LIN {X 0.019,Y -212.975,Z 813.838,A 0.000,B 0.000,C 90.000,E1 330.845} C_DIS
LIN {X 0.093,Y -220.835,Z 813.816,A 0.000,B 0.000,C 90.000,E1 326.914} C_DIS
LIN {X -0.032,Y -227.717,Z 813.799,A 0.000,B 0.000,C 90.000,E1 323.863} C_DIS
LIN {X 0.055,Y -235.033,Z 813.782,A 0.000,B 0.000,C 90.000,E1 320.803} C_DIS
LIN {X -0.068,Y -244.076,Z 813.764,A 0.000,B 0.000,C 90.000,E1 317.472} C_DIS
LIN {X -0.126,Y -253.936,Z 813.745,A 0.000,B 0.000,C 90.000,E1 314.190} C_DIS
LIN {X -0.103,Y -263.291,Z 813.729,A 0.000,B 0.000,C 90.000,E1 311.310} C_DIS
LIN {X 0.023,Y -275.912,Z 813.710,A 0.000,B 0.000,C 90.000,E1 307.764} C_DIS
LIN {X -0.077,Y -288.380,Z 813.693,A 0.000,B 0.000,C 90.000,E1 304.692} C_DIS
LIN {X -0.096,Y -300.556,Z 813.678,A 0.000,B 0.000,C 90.000,E1 302.005} C_DIS
LIN {X 0.089,Y -312.158,Z 813.665,A 0.000,B 0.000,C 90.000,E1 299.667} C_DIS
LIN {X -0.018,Y -328.621,Z 813.649,A 0.000,B 0.000,C 90.000,E1 296.796} C_DIS
LIN {X 0.198,Y -346.426,Z 813.633,A 0.000,B 0.000,C 90.000,E1 293.951} C_DIS
LIN {X 0.036,Y -359.385,Z 813.623,A 0.000,B 0.000,C 90.000,E1 292.153} C_DIS
LIN {X 0.081,Y -375.773,Z 813.612,A 0.000,B 0.000,C 90.000,E1 290.066} C_DIS
LIN {X -0.012,Y -393.420,Z 813.600,A 0.000,B 0.000,C 90.000,E1 288.055} C_DIS
LIN {X -0.013,Y -411.061,Z 813.590,A 0.000,B 0.000,C 90.000,E1 286.134} C_DIS
LIN {X 0.036,Y -423.562,Z 813.582,A 0.000,B 0.000,C 90.000,E1 284.773} C_DIS
LIN {X 0.129,Y -435.900,Z 813.575,A 0.000,B 0.000,C 90.000,E1 283.411} C_DIS
LIN {X 0.080,Y -445.463,Z 813.569,A 0.000,B 0.000,C 90.000,E1 282.355} C_DIS
LIN {X -0.139,Y -456.594,Z 813.561,A 0.000,B 0.000,C 90.000,E1 281.074} C_DIS
LIN {X 0.054,Y -464.756,Z 813.556,A 0.000,B 0.000,C 90.000,E1 280.018} C_DIS
LIN {X -0.204,Y -472.214,Z 813.550,A 0.000,B 0.000,C 90.000,E1 279.029} C_DIS
LIN {X 0.228,Y -477.257,Z 813.546,A 0.000,B 0.000,C 90.000,E1 278.219} C_DIS
LIN {X 0.169,Y -481.626,Z 813.542,A 0.000,B 0.000,C 90.000,E1 277.473} C_DIS
LIN {X 0.218,Y -485.397,Z 813.537,A 0.000,B 0.000,C 90.000,E1 276.720} C_DIS
LIN {X -0.195,Y -488.429,Z 813.533,A 0.000,B 0.000,C 90.000,E1 276.024} C_DIS
LIN {X -0.042,Y -490.064,Z 813.531,A 0.000,B 0.000,C 90.000,E1 275.511} C_DIS
LIN {X 0.172,Y -491.281,Z 813.528,A 0.000,B 0.000,C 90.000,E1 274.992} C_DIS
LIN {X -0.095,Y -492.106,Z 813.525,A 0.000,B 0.000,C 90.000,E1 274.531} C_DIS
LIN {X 0.133,Y -492.547,Z 813.522,A 0.000,B 0.000,C 90.000,E1 274.012} C_DIS
LIN {X -0.160,Y -492.648,Z 813.520,A 0.000,B 0.000,C 90.000,E1 273.555} C_DIS
LIN {X 0.072,Y -492.322,Z 813.517,A 0.000,B 0.000,C 90.000,E1 273.037} C_DIS
LIN {X -0.213,Y -491.589,Z 813.514,A 0.000,B 0.000,C 90.000,E1 272.579} C_DIS
LIN {X -0.007,Y -490.500,Z 813.511,A 0.000,B 0.000,C 90.000,E1 272.064} C_DIS
LIN {X 0.211,Y -488.923,Z 813.509,A 0.000,B 0.000,C 90.000,E1 271.547} C_DIS
LIN {X -0.082,Y -486.963,Z 813.506,A 0.000,B 0.000,C 90.000,E1 271.088} C_DIS
LIN {X 0.106,Y -484.457,Z 813.503,A 0.000,B 0.000,C 90.000,E1 270.573} C_DIS
LIN {X -0.207,Y -481.352,Z 813.500,A 0.000,B 0.000,C 90.000,E1 270.115} C_DIS
LIN {X -0.053,Y -477.541,Z 813.498,A 0.000,B 0.000,C 90.000,E1 269.599} C_DIS
LIN {X 0.077,Y -472.892,Z 813.495,A 0.000,B 0.000,C 90.000,E1 269.083} C_DIS
LIN {X 0.214,Y -467.213,Z 813.492,A 0.000,B 0.000,C 90.000,E1 268.568} C_DIS
LIN {X -0.189,Y -464.243,Z 813.491,A 0.000,B 0.000,C 90.000,E1 268.396} C_DIS
LIN {X -0.213,Y -457.716,Z 813.489,A 0.000,B 0.000,C 90.000,E1 267.993} C_DIS
LIN {X -0.131,Y -450.659,Z 813.487,A 0.000,B 0.000,C 90.000,E1 267.650} C_DIS
LIN {X 0.053,Y -442.949,Z 813.485,A 0.000,B 0.000,C 90.000,E1 267.364} C_DIS
LIN {X -0.148,Y -434.987,Z 813.484,A 0.000,B 0.000,C 90.000,E1 267.192} C_DIS
LIN {X 0.170,Y -427.099,Z 813.484,A 0.000,B 0.000,C 90.000,E1 267.020} C_DIS
LIN {X 0.184,Y -419.177,Z 813.483,A 0.000,B 0.000,C 90.000,E1 266.963} C_DIS
LIN {X 0.051,Y -180.989,Z 813.483,A 0.000,B 0.000,C 90.000,E1 266.963} C_DIS
LIN {X -0.017,Y -180.848,Z 813.472,A 0.000,B 0.000,C 90.000,E1 264.951} C_DIS
LIN {X 0.066,Y -178.958,Z 813.444,A 0.000,B 0.000,C 90.000,E1 259.859} C_DIS
LIN {X -0.043,Y -177.363,Z 813.430,A 0.000,B 0.000,C 90.000,E1 257.353} C_DIS
LIN {X 0.053,Y -175.535,Z 813.411,A 0.000,B 0.000,C 90.000,E1 253.921} C_DIS
LIN {X 0.054,Y -172.270,Z 813.387,A 0.000,B 0.000,C 90.000,E1 249.645} C_DIS
LIN {X 0.093,Y -171.749,Z 813.382,A 0.000,B 0.000,C 90.000,E1 248.773} C_DIS
LIN {X -0.050,Y -167.346,Z 813.353,A 0.000,B 0.000,C 90.000,E1 243.640} C_DIS
LIN {X 0.032,Y -166.734,Z 813.349,A 0.000,B 0.000,C 90.000,E1 242.743} C_DIS
LIN {X -0.055,Y -162.714,Z 813.324,A 0.000,B 0.000,C 90.000,E1 238.408} C_DIS
LIN {X 0.006,Y -161.404,Z 813.315,A 0.000,B 0.000,C 90.000,E1 236.628} C_DIS
LIN {X 0.048,Y -157.396,Z 813.290,A 0.000,B 0.000,C 90.000,E1 232.190} C_DIS
LIN {X -0.019,Y -155.394,Z 813.275,A 0.000,B 0.000,C 90.000,E1 229.542} C_DIS
LIN {X 0.021,Y -151.727,Z 813.250,A 0.000,B 0.000,C 90.000,E1 225.040} C_DIS
LIN {X 0.037,Y -149.923,Z 813.235,A 0.000,B 0.000,C 90.000,E1 222.324} C_DIS
LIN {X -0.046,Y -146.775,Z 813.210,A 0.000,B 0.000,C 90.000,E1 217.810} C_DIS
LIN {X 0.058,Y -145.346,Z 813.195,A 0.000,B 0.000,C 90.000,E1 215.025} C_DIS
LIN {X -0.027,Y -142.420,Z 813.164,A 0.000,B 0.000,C 90.000,E1 209.539} C_DIS
LIN {X 0.022,Y -141.407,Z 813.149,A 0.000,B 0.000,C 90.000,E1 206.744} C_DIS
LIN {X 0.009,Y -139.358,Z 813.112,A 0.000,B 0.000,C 90.000,E1 200.248} C_DIS
LIN {X -0.002,Y -138.799,Z 813.097,A 0.000,B 0.000,C 90.000,E1 197.457} C_DIS
LIN {X 0.052,Y -138.348,Z 813.055,A 0.000,B 0.000,C 90.000,E1 189.962} C_DIS
LIN {X 0.070,Y -139.370,Z 813.009,A 0.000,B 0.000,C 90.000,E1 181.547} C_DIS
LIN {X -0.016,Y -141.258,Z 812.973,A 0.000,B 0.000,C 90.000,E1 175.065} C_DIS
LIN {X -0.058,Y -142.626,Z 812.957,A 0.000,B 0.000,C 90.000,E1 172.299} C_DIS
LIN {X 0.035,Y -144.948,Z 812.931,A 0.000,B 0.000,C 90.000,E1 167.645} C_DIS
LIN {X 0.026,Y -147.577,Z 812.911,A 0.000,B 0.000,C 90.000,E1 163.976} C_DIS
LIN {X -0.085,Y -150.189,Z 812.891,A 0.000,B 0.000,C 90.000,E1 160.369} C_DIS
LIN {X -0.077,Y -153.568,Z 812.871,A 0.000,B 0.000,C 90.000,E1 156.741} C_DIS
LIN {X -0.026,Y -156.985,Z 812.851,A 0.000,B 0.000,C 90.000,E1 153.127} C_DIS
LIN {X 0.047,Y -161.098,Z 812.831,A 0.000,B 0.000,C 90.000,E1 149.537} C_DIS
LIN {X -0.007,Y -163.201,Z 812.821,A 0.000,B 0.000,C 90.000,E1 147.788} C_DIS
LIN {X -0.002,Y -167.628,Z 812.802,A 0.000,B 0.000,C 90.000,E1 144.276} C_DIS
LIN {X 0.013,Y -171.455,Z 812.787,A 0.000,B 0.000,C 90.000,E1 141.662} C_DIS
LIN {X -0.056,Y -176.379,Z 812.768,A 0.000,B 0.000,C 90.000,E1 138.243} C_DIS
LIN {X 0.066,Y -180.671,Z 812.754,A 0.000,B 0.000,C 90.000,E1 135.648} C_DIS
LIN {X 0.048,Y -186.074,Z 812.735,A 0.000,B 0.000,C 90.000,E1 132.285} C_DIS
LIN {X -0.015,Y -190.711,Z 812.721,A 0.000,B 0.000,C 90.000,E1 129.806} C_DIS
LIN {X 0.035,Y -192.711,Z 812.714,A 0.000,B 0.000,C 90.000,E1 128.588} C_DIS
LIN {X 0.010,Y -293.159,Z 812.714,A 0.000,B 0.000,C 90.000,E1 128.588} C_DIS
LIN {X -0.075,Y -294.254,Z 812.714,A 0.000,B 0.000,C 90.000,E1 128.588} C_DIS
LIN {X -0.110,Y -299.039,Z 812.713,A 0.000,B 0.000,C 90.000,E1 128.382} C_DIS
LIN {X -0.143,Y -301.560,Z 812.712,A 0.000,B 0.000,C 90.000,E1 128.177} C_DIS
LIN {X 0.042,Y -305.369,Z 812.709,A 0.000,B 0.000,C 90.000,E1 127.649} C_DIS
LIN {X 0.053,Y -307.140,Z 812.707,A 0.000,B 0.000,C 90.000,E1 127.317} C_DIS
LIN {X 0.006,Y -308.524,Z 812.706,A 0.000,B 0.000,C 90.000,E1 126.996} C_DIS
LIN {X -0.054,Y -316.443,Z 812.691,A 0.000,B 0.000,C 90.000,E1 124.405} C_DIS
LIN {X -0.054,Y -327.496,Z 812.673,A 0.000,B 0.000,C 90.000,E1 121.209} C_DIS
LIN {X 0.114,Y -338.834,Z 812.658,A 0.000,B 0.000,C 90.000,E1 118.359} C_DIS
LIN {X 0.122,Y -351.598,Z 812.642,A 0.000,B 0.000,C 90.000,E1 115.591} C_DIS
LIN {X -0.026,Y -364.229,Z 812.629,A 0.000,B 0.000,C 90.000,E1 113.206} C_DIS
LIN {X -0.008,Y -378.165,Z 812.616,A 0.000,B 0.000,C 90.000,E1 110.844} C_DIS
LIN {X -0.045,Y -393.504,Z 812.603,A 0.000,B 0.000,C 90.000,E1 108.544} C_DIS
LIN {X 0.190,Y -410.357,Z 812.590,A 0.000,B 0.000,C 90.000,E1 106.260} C_DIS
LIN {X -0.190,Y -428.847,Z 812.578,A 0.000,B 0.000,C 90.000,E1 104.120} C_DIS
LIN {X -0.052,Y -448.726,Z 812.567,A 0.000,B 0.000,C 90.000,E1 102.007} C_DIS
LIN {X -0.001,Y -466.598,Z 812.557,A 0.000,B 0.000,C 90.000,E1 100.310} C_DIS
LIN {X 0.023,Y -468.920,Z 812.556,A 0.000,B 0.000,C 90.000,E1 100.074} C_DIS
LIN {X -0.160,Y -470.769,Z 812.555,A 0.000,B 0.000,C 90.000,E1 99.849} C_DIS
LIN {X 0.202,Y -472.166,Z 812.553,A 0.000,B 0.000,C 90.000,E1 99.557} C_DIS
LIN {X -0.163,Y -473.990,Z 812.550,A 0.000,B 0.000,C 90.000,E1 99.095} C_DIS
LIN {X 0.022,Y -474.720,Z 812.548,A 0.000,B 0.000,C 90.000,E1 98.568} C_DIS
LIN {X 0.146,Y -474.481,Z 812.545,A 0.000,B 0.000,C 90.000,E1 98.049} C_DIS
LIN {X -0.193,Y -473.242,Z 812.542,A 0.000,B 0.000,C 90.000,E1 97.587} C_DIS
LIN {X 0.136,Y -472.188,Z 812.541,A 0.000,B 0.000,C 90.000,E1 97.296} C_DIS
LIN {X -0.063,Y -470.775,Z 812.539,A 0.000,B 0.000,C 90.000,E1 97.068} C_DIS
LIN {X 0.086,Y -453.158,Z 812.524,A 0.000,B 0.000,C 90.000,E1 94.245} C_DIS
LIN {X 0.028,Y -444.098,Z 812.515,A 0.000,B 0.000,C 90.000,E1 92.694} C_DIS
LIN {X -0.045,Y -433.373,Z 812.505,A 0.000,B 0.000,C 90.000,E1 90.859} C_DIS
LIN {X -0.041,Y -423.794,Z 812.496,A 0.000,B 0.000,C 90.000,E1 89.255} C_DIS
LIN {X -0.192,Y -414.104,Z 812.487,A 0.000,B 0.000,C 90.000,E1 87.650} C_DIS
LIN {X -0.104,Y -404.224,Z 812.478,A 0.000,B 0.000,C 90.000,E1 85.988} C_DIS
LIN {X -0.056,Y -391.053,Z 812.465,A 0.000,B 0.000,C 90.000,E1 83.742} C_DIS
LIN {X 0.110,Y -378.181,Z 812.453,A 0.000,B 0.000,C 90.000,E1 81.432} C_DIS
LIN {X 0.059,Y -364.163,Z 812.438,A 0.000,B 0.000,C 90.000,E1 78.814} C_DIS
LIN {X 0.132,Y -350.810,Z 812.423,A 0.000,B 0.000,C 90.000,E1 76.117} C_DIS
LIN {X -0.134,Y -340.550,Z 812.411,A 0.000,B 0.000,C 90.000,E1 74.031} C_DIS
LIN {X 0.111,Y -328.959,Z 812.397,A 0.000,B 0.000,C 90.000,E1 71.511} C_DIS
LIN {X 0.091,Y -316.298,Z 812.382,A 0.000,B 0.000,C 90.000,E1 68.666} C_DIS
LIN {X 0.067,Y -302.768,Z 812.364,A 0.000,B 0.000,C 90.000,E1 65.433} C_DIS
LIN {X -0.116,Y -290.215,Z 812.345,A 0.000,B 0.000,C 90.000,E1 62.153} C_DIS
LIN {X 0.070,Y -280.606,Z 812.330,A 0.000,B 0.000,C 90.000,E1 59.410} C_DIS
LIN {X 0.127,Y -270.334,Z 812.313,A 0.000,B 0.000,C 90.000,E1 56.294} C_DIS
LIN {X 0.016,Y -262.692,Z 812.299,A 0.000,B 0.000,C 90.000,E1 53.863} C_DIS
LIN {X -0.023,Y -256.222,Z 812.287,A 0.000,B 0.000,C 90.000,E1 51.743} C_DIS
LIN {X -0.135,Y -245.708,Z 812.267,A 0.000,B 0.000,C 90.000,E1 48.162} C_DIS
LIN {X 0.059,Y -235.971,Z 812.247,A 0.000,B 0.000,C 90.000,E1 44.433} C_DIS
LIN {X 0.061,Y -228.787,Z 812.230,A 0.000,B 0.000,C 90.000,E1 41.434} C_DIS
LIN {X 0.091,Y -221.797,Z 812.213,A 0.000,B 0.000,C 90.000,E1 38.382} C_DIS
LIN {X 0.027,Y -215.062,Z 812.196,A 0.000,B 0.000,C 90.000,E1 35.311} C_DIS
LIN {X -0.092,Y -208.765,Z 812.179,A 0.000,B 0.000,C 90.000,E1 32.212} C_DIS
LIN {X 0.050,Y -203.122,Z 812.161,A 0.000,B 0.000,C 90.000,E1 28.999} C_DIS
LIN {X 0.016,Y -198.116,Z 812.143,A 0.000,B 0.000,C 90.000,E1 25.796} C_DIS
LIN {X 0.068,Y -192.972,Z 812.121,A 0.000,B 0.000,C 90.000,E1 21.716} C_DIS
LIN {X -0.032,Y -188.939,Z 812.098,A 0.000,B 0.000,C 90.000,E1 17.638} C_DIS
LIN {X 0.015,Y -185.716,Z 812.070,A 0.000,B 0.000,C 90.000,E1 12.647} C_DIS
LIN {X 0.081,Y -183.567,Z 812.029,A 0.000,B 0.000,C 90.000,E1 5.106} C_DIS
LIN {X -0.018,Y -185.536,Z 811.974,A 0.000,B 0.000,C 90.000,E1 355.355} C_DIS
LIN {X 0.074,Y -188.490,Z 811.946,A 0.000,B 0.000,C 90.000,E1 350.330} C_DIS
LIN {X -0.051,Y -192.670,Z 811.919,A 0.000,B 0.000,C 90.000,E1 345.408} C_DIS
LIN {X 0.075,Y -197.155,Z 811.896,A 0.000,B 0.000,C 90.000,E1 341.275} C_DIS
LIN {X 0.046,Y -202.557,Z 811.874,A 0.000,B 0.000,C 90.000,E1 337.230} C_DIS
LIN {X -0.060,Y -208.856,Z 811.851,A 0.000,B 0.000,C 90.000,E1 333.256} C_DIS
LIN {X -0.007,Y -214.686,Z 811.834,A 0.000,B 0.000,C 90.000,E1 330.078} C_DIS
LIN {X 0.042,Y -222.708,Z 811.812,A 0.000,B 0.000,C 90.000,E1 326.167} C_DIS
LIN {X -0.019,Y -231.471,Z 811.791,A 0.000,B 0.000,C 90.000,E1 322.351} C_DIS
LIN {X 0.108,Y -240.106,Z 811.772,A 0.000,B 0.000,C 90.000,E1 318.933} C_DIS
LIN {X 0.123,Y -250.644,Z 811.752,A 0.000,B 0.000,C 90.000,E1 315.243} C_DIS
LIN {X 0.055,Y -259.822,Z 811.735,A 0.000,B 0.000,C 90.000,E1 312.366} C_DIS
LIN {X -0.051,Y -270.794,Z 811.718,A 0.000,B 0.000,C 90.000,E1 309.197} C_DIS
LIN {X -0.141,Y -282.654,Z 811.700,A 0.000,B 0.000,C 90.000,E1 306.091} C_DIS
LIN {X 0.002,Y -297.359,Z 811.682,A 0.000,B 0.000,C 90.000,E1 302.673} C_DIS
LIN {X 0.194,Y -312.076,Z 811.665,A 0.000,B 0.000,C 90.000,E1 299.667} C_DIS
LIN {X -0.057,Y -328.518,Z 811.649,A 0.000,B 0.000,C 90.000,E1 296.821} C_DIS
LIN {X -0.007,Y -346.258,Z 811.633,A 0.000,B 0.000,C 90.000,E1 294.003} C_DIS
LIN {X -0.132,Y -361.417,Z 811.622,A 0.000,B 0.000,C 90.000,E1 291.897} C_DIS
LIN {X -0.063,Y -377.967,Z 811.610,A 0.000,B 0.000,C 90.000,E1 289.812} C_DIS
LIN {X 0.099,Y -393.111,Z 811.600,A 0.000,B 0.000,C 90.000,E1 288.055} C_DIS
LIN {X -0.065,Y -410.914,Z 811.590,A 0.000,B 0.000,C 90.000,E1 286.134} C_DIS
LIN {X 0.041,Y -423.321,Z 811.582,A 0.000,B 0.000,C 90.000,E1 284.773} C_DIS
LIN {X 0.130,Y -435.663,Z 811.575,A 0.000,B 0.000,C 90.000,E1 283.411} C_DIS
LIN {X 0.078,Y -445.225,Z 811.569,A 0.000,B 0.000,C 90.000,E1 282.355} C_DIS
LIN {X -0.144,Y -456.367,Z 811.561,A 0.000,B 0.000,C 90.000,E1 281.074} C_DIS
LIN {X 0.046,Y -464.508,Z 811.556,A 0.000,B 0.000,C 90.000,E1 280.018} C_DIS
LIN {X 0.252,Y -472.006,Z 811.550,A 0.000,B 0.000,C 90.000,E1 278.973} C_DIS
LIN {X 0.215,Y -477.096,Z 811.546,A 0.000,B 0.000,C 90.000,E1 278.219} C_DIS
LIN {X 0.155,Y -481.476,Z 811.542,A 0.000,B 0.000,C 90.000,E1 277.473} C_DIS
LIN {X 0.201,Y -485.253,Z 811.537,A 0.000,B 0.000,C 90.000,E1 276.720} C_DIS
LIN {X -0.213,Y -488.319,Z 811.533,A 0.000,B 0.000,C 90.000,E1 276.024} C_DIS
LIN {X -0.061,Y -489.972,Z 811.531,A 0.000,B 0.000,C 90.000,E1 275.511} C_DIS
LIN {X 0.153,Y -491.224,Z 811.528,A 0.000,B 0.000,C 90.000,E1 274.992} C_DIS
LIN {X -0.114,Y -492.070,Z 811.525,A 0.000,B 0.000,C 90.000,E1 274.531} C_DIS
LIN {X 0.113,Y -492.553,Z 811.522,A 0.000,B 0.000,C 90.000,E1 274.012} C_DIS
LIN {X -0.180,Y -492.634,Z 811.520,A 0.000,B 0.000,C 90.000,E1 273.555} C_DIS
LIN {X 0.051,Y -492.328,Z 811.517,A 0.000,B 0.000,C 90.000,E1 273.037} C_DIS
LIN {X -0.234,Y -491.607,Z 811.514,A 0.000,B 0.000,C 90.000,E1 272.579} C_DIS
LIN {X -0.027,Y -490.491,Z 811.511,A 0.000,B 0.000,C 90.000,E1 272.064} C_DIS
LIN {X 0.191,Y -488.982,Z 811.509,A 0.000,B 0.000,C 90.000,E1 271.547} C_DIS
LIN {X -0.101,Y -487.021,Z 811.506,A 0.000,B 0.000,C 90.000,E1 271.088} C_DIS
LIN {X 0.087,Y -484.536,Z 811.503,A 0.000,B 0.000,C 90.000,E1 270.573} C_DIS
LIN {X -0.226,Y -481.466,Z 811.500,A 0.000,B 0.000,C 90.000,E1 270.115} C_DIS
LIN {X -0.072,Y -477.698,Z 811.498,A 0.000,B 0.000,C 90.000,E1 269.599} C_DIS
LIN {X 0.061,Y -473.104,Z 811.495,A 0.000,B 0.000,C 90.000,E1 269.083} C_DIS
LIN {X 0.165,Y -467.429,Z 811.492,A 0.000,B 0.000,C 90.000,E1 268.568} C_DIS
LIN {X 0.223,Y -464.498,Z 811.491,A 0.000,B 0.000,C 90.000,E1 268.339} C_DIS
LIN {X -0.166,Y -461.181,Z 811.490,A 0.000,B 0.000,C 90.000,E1 268.165} C_DIS
LIN {X 0.032,Y -454.214,Z 811.488,A 0.000,B 0.000,C 90.000,E1 267.764} C_DIS
LIN {X -0.087,Y -446.786,Z 811.486,A 0.000,B 0.000,C 90.000,E1 267.478} C_DIS
LIN {X -0.117,Y -438.709,Z 811.485,A 0.000,B 0.000,C 90.000,E1 267.249} C_DIS
LIN {X -0.104,Y -430.124,Z 811.484,A 0.000,B 0.000,C 90.000,E1 267.078} C_DIS
LIN {X 0.144,Y -422.727,Z 811.483,A 0.000,B 0.000,C 90.000,E1 266.963} C_DIS
LIN {X 0.011,Y -417.757,Z 811.483,A 0.000,B 0.000,C 90.000,E1 266.963} C_DIS
LIN {X -0.024,Y -180.987,Z 811.483,A 0.000,B 0.000,C 90.000,E1 266.963} C_DIS
LIN {X 0.090,Y -180.843,Z 811.472,A 0.000,B 0.000,C 90.000,E1 264.894} C_DIS
LIN {X -0.008,Y -178.951,Z 811.444,A 0.000,B 0.000,C 90.000,E1 259.859} C_DIS
LIN {X 0.009,Y -176.856,Z 811.425,A 0.000,B 0.000,C 90.000,E1 256.464} C_DIS
LIN {X -0.019,Y -175.516,Z 811.411,A 0.000,B 0.000,C 90.000,E1 253.921} C_DIS
LIN {X -0.017,Y -172.254,Z 811.387,A 0.000,B 0.000,C 90.000,E1 249.645} C_DIS
LIN {X 0.022,Y -171.733,Z 811.382,A 0.000,B 0.000,C 90.000,E1 248.773} C_DIS
LIN {X 0.031,Y -167.330,Z 811.353,A 0.000,B 0.000,C 90.000,E1 243.589} C_DIS
LIN {X -0.038,Y -166.714,Z 811.349,A 0.000,B 0.000,C 90.000,E1 242.743} C_DIS
LIN {X 0.100,Y -162.694,Z 811.324,A 0.000,B 0.000,C 90.000,E1 238.329} C_DIS
LIN {X -0.061,Y -161.385,Z 811.314,A 0.000,B 0.000,C 90.000,E1 236.628} C_DIS
LIN {X -0.019,Y -157.378,Z 811.290,A 0.000,B 0.000,C 90.000,E1 232.190} C_DIS
LIN {X -0.086,Y -155.371,Z 811.275,A 0.000,B 0.000,C 90.000,E1 229.542} C_DIS
LIN {X 0.062,Y -151.711,Z 811.250,A 0.000,B 0.000,C 90.000,E1 225.000} C_DIS
LIN {X -0.029,Y -149.902,Z 811.235,A 0.000,B 0.000,C 90.000,E1 222.324} C_DIS
LIN {X 0.096,Y -146.761,Z 811.210,A 0.000,B 0.000,C 90.000,E1 217.729} C_DIS
LIN {X -0.007,Y -145.329,Z 811.195,A 0.000,B 0.000,C 90.000,E1 215.025} C_DIS
LIN {X 0.033,Y -142.410,Z 811.164,A 0.000,B 0.000,C 90.000,E1 209.489} C_DIS
LIN {X -0.041,Y -141.395,Z 811.148,A 0.000,B 0.000,C 90.000,E1 206.744} C_DIS
LIN {X -0.053,Y -139.354,Z 811.112,A 0.000,B 0.000,C 90.000,E1 200.248} C_DIS
LIN {X -0.064,Y -138.793,Z 811.097,A 0.000,B 0.000,C 90.000,E1 197.457} C_DIS
LIN {X -0.010,Y -138.347,Z 811.055,A 0.000,B 0.000,C 90.000,E1 189.962} C_DIS
LIN {X 0.007,Y -139.378,Z 811.009,A 0.000,B 0.000,C 90.000,E1 181.547} C_DIS
LIN {X 0.061,Y -141.270,Z 810.972,A 0.000,B 0.000,C 90.000,E1 175.008} C_DIS
LIN {X 0.019,Y -142.636,Z 810.957,A 0.000,B 0.000,C 90.000,E1 172.243} C_DIS
LIN {X -0.029,Y -144.964,Z 810.931,A 0.000,B 0.000,C 90.000,E1 167.645} C_DIS
LIN {X -0.039,Y -147.592,Z 810.911,A 0.000,B 0.000,C 90.000,E1 163.976} C_DIS
LIN {X -0.009,Y -150.209,Z 810.891,A 0.000,B 0.000,C 90.000,E1 160.315} C_DIS
LIN {X 0.058,Y -153.594,Z 810.870,A 0.000,B 0.000,C 90.000,E1 156.666} C_DIS
LIN {X 0.047,Y -157.010,Z 810.851,A 0.000,B 0.000,C 90.000,E1 153.076} C_DIS
LIN {X -0.021,Y -161.129,Z 810.831,A 0.000,B 0.000,C 90.000,E1 149.537} C_DIS
LIN {X -0.076,Y -163.229,Z 810.821,A 0.000,B 0.000,C 90.000,E1 147.788} C_DIS
LIN {X -0.073,Y -167.662,Z 810.801,A 0.000,B 0.000,C 90.000,E1 144.276} C_DIS
LIN {X 0.076,Y -171.486,Z 810.787,A 0.000,B 0.000,C 90.000,E1 141.618} C_DIS
LIN {X 0.120,Y -176.416,Z 810.768,A 0.000,B 0.000,C 90.000,E1 138.162} C_DIS
LIN {X -0.008,Y -180.710,Z 810.754,A 0.000,B 0.000,C 90.000,E1 135.648} C_DIS
LIN {X -0.027,Y -186.114,Z 810.735,A 0.000,B 0.000,C 90.000,E1 132.285} C_DIS
LIN {X 0.031,Y -190.752,Z 810.721,A 0.000,B 0.000,C 90.000,E1 129.769} C_DIS
LIN {X -0.039,Y -192.687,Z 810.715,A 0.000,B 0.000,C 90.000,E1 128.624} C_DIS
LIN {X -0.094,Y -292.430,Z 810.714,A 0.000,B 0.000,C 90.000,E1 128.624} C_DIS
LIN {X 0.041,Y -295.443,Z 810.714,A 0.000,B 0.000,C 90.000,E1 128.543} C_DIS
LIN {X 0.008,Y -299.450,Z 810.713,A 0.000,B 0.000,C 90.000,E1 128.338} C_DIS
LIN {X 0.161,Y -301.838,Z 810.712,A 0.000,B 0.000,C 90.000,E1 128.096} C_DIS
LIN {X 0.039,Y -305.657,Z 810.709,A 0.000,B 0.000,C 90.000,E1 127.604} C_DIS
LIN {X -0.007,Y -307.351,Z 810.707,A 0.000,B 0.000,C 90.000,E1 127.282} C_DIS
LIN {X 0.007,Y -308.678,Z 810.705,A 0.000,B 0.000,C 90.000,E1 126.950} C_DIS
LIN {X -0.117,Y -320.807,Z 810.684,A 0.000,B 0.000,C 90.000,E1 123.086} C_DIS
LIN {X 0.016,Y -331.274,Z 810.668,A 0.000,B 0.000,C 90.000,E1 120.207} C_DIS
LIN {X 0.126,Y -343.099,Z 810.652,A 0.000,B 0.000,C 90.000,E1 117.385} C_DIS
LIN {X 0.106,Y -356.382,Z 810.637,A 0.000,B 0.000,C 90.000,E1 114.643} C_DIS
LIN {X -0.066,Y -369.514,Z 810.624,A 0.000,B 0.000,C 90.000,E1 112.280} C_DIS
LIN {X -0.050,Y -383.987,Z 810.611,A 0.000,B 0.000,C 90.000,E1 109.939} C_DIS
LIN {X 0.065,Y -399.906,Z 810.598,A 0.000,B 0.000,C 90.000,E1 107.638} C_DIS
LIN {X -0.051,Y -417.386,Z 810.586,A 0.000,B 0.000,C 90.000,E1 105.426} C_DIS
LIN {X 0.069,Y -436.527,Z 810.574,A 0.000,B 0.000,C 90.000,E1 103.244} C_DIS
LIN {X -0.131,Y -456.663,Z 810.562,A 0.000,B 0.000,C 90.000,E1 101.243} C_DIS
LIN {X 0.187,Y -466.939,Z 810.557,A 0.000,B 0.000,C 90.000,E1 100.254} C_DIS
LIN {X 0.215,Y -469.175,Z 810.556,A 0.000,B 0.000,C 90.000,E1 100.018} C_DIS
LIN {X -0.011,Y -470.993,Z 810.554,A 0.000,B 0.000,C 90.000,E1 99.792} C_DIS
LIN {X -0.158,Y -472.359,Z 810.553,A 0.000,B 0.000,C 90.000,E1 99.557} C_DIS
LIN {X 0.020,Y -474.085,Z 810.550,A 0.000,B 0.000,C 90.000,E1 99.029} C_DIS
LIN {X 0.134,Y -474.734,Z 810.547,A 0.000,B 0.000,C 90.000,E1 98.511} C_DIS
LIN {X -0.212,Y -474.418,Z 810.545,A 0.000,B 0.000,C 90.000,E1 98.049} C_DIS
LIN {X -0.081,Y -473.091,Z 810.542,A 0.000,B 0.000,C 90.000,E1 97.530} C_DIS
LIN {X -0.220,Y -471.985,Z 810.540,A 0.000,B 0.000,C 90.000,E1 97.296} C_DIS
LIN {X -0.099,Y -468.842,Z 810.538,A 0.000,B 0.000,C 90.000,E1 96.777} C_DIS
LIN {X -0.013,Y -451.408,Z 810.522,A 0.000,B 0.000,C 90.000,E1 93.955} C_DIS
LIN {X 0.056,Y -440.816,Z 810.512,A 0.000,B 0.000,C 90.000,E1 92.121} C_DIS
LIN {X 0.198,Y -431.549,Z 810.503,A 0.000,B 0.000,C 90.000,E1 90.516} C_DIS
LIN {X 0.165,Y -421.945,Z 810.494,A 0.000,B 0.000,C 90.000,E1 88.912} C_DIS
LIN {X -0.024,Y -412.251,Z 810.485,A 0.000,B 0.000,C 90.000,E1 87.306} C_DIS
LIN {X 0.052,Y -402.336,Z 810.476,A 0.000,B 0.000,C 90.000,E1 85.641} C_DIS
LIN {X 0.059,Y -389.212,Z 810.463,A 0.000,B 0.000,C 90.000,E1 83.394} C_DIS
LIN {X 0.180,Y -376.401,Z 810.451,A 0.000,B 0.000,C 90.000,E1 81.084} C_DIS
LIN {X 0.054,Y -360.966,Z 810.434,A 0.000,B 0.000,C 90.000,E1 78.173} C_DIS
LIN {X 0.120,Y -347.729,Z 810.419,A 0.000,B 0.000,C 90.000,E1 75.463} C_DIS
LIN {X 0.118,Y -337.479,Z 810.407,A 0.000,B 0.000,C 90.000,E1 73.323} C_DIS
LIN {X -0.043,Y -325.958,Z 810.394,A 0.000,B 0.000,C 90.000,E1 70.859} C_DIS
LIN {X 0.147,Y -314.805,Z 810.380,A 0.000,B 0.000,C 90.000,E1 68.284} C_DIS
LIN {X 0.102,Y -300.155,Z 810.360,A 0.000,B 0.000,C 90.000,E1 64.717} C_DIS
LIN {X -0.139,Y -288.992,Z 810.343,A 0.000,B 0.000,C 90.000,E1 61.769} C_DIS
LIN {X 0.157,Y -279.494,Z 810.328,A 0.000,B 0.000,C 90.000,E1 58.997} C_DIS
LIN {X -0.119,Y -270.464,Z 810.313,A 0.000,B 0.000,C 90.000,E1 56.294} C_DIS
LIN {X -0.059,Y -262.850,Z 810.299,A 0.000,B 0.000,C 90.000,E1 53.829} C_DIS
LIN {X -0.042,Y -256.408,Z 810.287,A 0.000,B 0.000,C 90.000,E1 51.698} C_DIS
LIN {X 0.003,Y -247.959,Z 810.271,A 0.000,B 0.000,C 90.000,E1 48.809} C_DIS
LIN {X -0.080,Y -238.084,Z 810.251,A 0.000,B 0.000,C 90.000,E1 45.162} C_DIS
LIN {X 0.052,Y -229.017,Z 810.230,A 0.000,B 0.000,C 90.000,E1 41.391} C_DIS
LIN {X -0.078,Y -222.038,Z 810.213,A 0.000,B 0.000,C 90.000,E1 38.382} C_DIS
LIN {X 0.048,Y -213.656,Z 810.192,A 0.000,B 0.000,C 90.000,E1 34.485} C_DIS
LIN {X 0.072,Y -207.547,Z 810.174,A 0.000,B 0.000,C 90.000,E1 31.337} C_DIS
LIN {X 0.076,Y -202.045,Z 810.157,A 0.000,B 0.000,C 90.000,E1 28.153} C_DIS
LIN {X 0.014,Y -197.240,Z 810.139,A 0.000,B 0.000,C 90.000,E1 24.951} C_DIS
LIN {X 0.064,Y -192.351,Z 810.116,A 0.000,B 0.000,C 90.000,E1 20.865} C_DIS
LIN {X -0.113,Y -188.528,Z 810.093,A 0.000,B 0.000,C 90.000,E1 16.804} C_DIS
LIN {X 0.062,Y -185.577,Z 810.065,A 0.000,B 0.000,C 90.000,E1 11.771} C_DIS
LIN {X 0.093,Y -186.157,Z 809.970,A 0.000,B 0.000,C 90.000,E1 354.489} C_DIS
LIN {X 0.059,Y -189.316,Z 809.942,A 0.000,B 0.000,C 90.000,E1 349.511} C_DIS
LIN {X -0.027,Y -192.867,Z 809.919,A 0.000,B 0.000,C 90.000,E1 345.408} C_DIS
LIN {X 0.105,Y -197.312,Z 809.896,A 0.000,B 0.000,C 90.000,E1 341.275} C_DIS
LIN {X 0.082,Y -202.702,Z 809.874,A 0.000,B 0.000,C 90.000,E1 337.230} C_DIS
LIN {X 0.081,Y -207.667,Z 809.856,A 0.000,B 0.000,C 90.000,E1 334.024} C_DIS
LIN {X 0.008,Y -213.337,Z 809.838,A 0.000,B 0.000,C 90.000,E1 330.873} C_DIS
LIN {X 0.016,Y -221.210,Z 809.816,A 0.000,B 0.000,C 90.000,E1 326.962} C_DIS
LIN {X -0.032,Y -229.836,Z 809.795,A 0.000,B 0.000,C 90.000,E1 323.130} C_DIS
LIN {X -0.069,Y -237.280,Z 809.778,A 0.000,B 0.000,C 90.000,E1 320.114} C_DIS
LIN {X 0.045,Y -246.478,Z 809.760,A 0.000,B 0.000,C 90.000,E1 316.743} C_DIS
LIN {X 0.064,Y -256.446,Z 809.742,A 0.000,B 0.000,C 90.000,E1 313.461} C_DIS
LIN {X 0.039,Y -267.096,Z 809.724,A 0.000,B 0.000,C 90.000,E1 310.253} C_DIS
LIN {X -0.101,Y -279.964,Z 809.704,A 0.000,B 0.000,C 90.000,E1 306.790} C_DIS
LIN {X -0.035,Y -292.758,Z 809.687,A 0.000,B 0.000,C 90.000,E1 303.706} C_DIS
LIN {X -0.052,Y -308.587,Z 809.669,A 0.000,B 0.000,C 90.000,E1 300.384} C_DIS
LIN {X 0.100,Y -326.497,Z 809.651,A 0.000,B 0.000,C 90.000,E1 297.129} C_DIS
LIN {X -0.041,Y -346.100,Z 809.633,A 0.000,B 0.000,C 90.000,E1 294.027} C_DIS
LIN {X -0.025,Y -361.191,Z 809.622,A 0.000,B 0.000,C 90.000,E1 291.897} C_DIS
LIN {X 0.045,Y -377.713,Z 809.610,A 0.000,B 0.000,C 90.000,E1 289.812} C_DIS
LIN {X 0.238,Y -392.753,Z 809.601,A 0.000,B 0.000,C 90.000,E1 288.055} C_DIS
LIN {X 0.093,Y -410.507,Z 809.590,A 0.000,B 0.000,C 90.000,E1 286.134} C_DIS
LIN {X 0.188,Y -422.909,Z 809.582,A 0.000,B 0.000,C 90.000,E1 284.773} C_DIS
LIN {X -0.150,Y -435.258,Z 809.575,A 0.000,B 0.000,C 90.000,E1 283.467} C_DIS
LIN {X 0.221,Y -444.811,Z 809.569,A 0.000,B 0.000,C 90.000,E1 282.355} C_DIS
LIN {X -0.255,Y -453.816,Z 809.563,A 0.000,B 0.000,C 90.000,E1 281.366} C_DIS
LIN {X -0.096,Y -462.167,Z 809.557,A 0.000,B 0.000,C 90.000,E1 280.310} C_DIS
LIN {X 0.080,Y -469.842,Z 809.552,A 0.000,B 0.000,C 90.000,E1 279.265} C_DIS
LIN {X 0.019,Y -475.162,Z 809.547,A 0.000,B 0.000,C 90.000,E1 278.511} C_DIS
LIN {X 0.008,Y -479.833,Z 809.543,A 0.000,B 0.000,C 90.000,E1 277.757} C_DIS
LIN {X 0.032,Y -483.864,Z 809.539,A 0.000,B 0.000,C 90.000,E1 277.004} C_DIS
LIN {X 0.210,Y -486.153,Z 809.536,A 0.000,B 0.000,C 90.000,E1 276.486} C_DIS
LIN {X -0.133,Y -488.164,Z 809.533,A 0.000,B 0.000,C 90.000,E1 276.030} C_DIS
LIN {X 0.069,Y -489.807,Z 809.531,A 0.000,B 0.000,C 90.000,E1 275.511} C_DIS
LIN {X -0.207,Y -491.098,Z 809.528,A 0.000,B 0.000,C 90.000,E1 275.049} C_DIS
LIN {X 0.015,Y -492.001,Z 809.525,A 0.000,B 0.000,C 90.000,E1 274.531} C_DIS
LIN {X 0.241,Y -492.497,Z 809.522,A 0.000,B 0.000,C 90.000,E1 274.012} C_DIS
LIN {X -0.053,Y -492.617,Z 809.520,A 0.000,B 0.000,C 90.000,E1 273.555} C_DIS
LIN {X 0.179,Y -492.299,Z 809.517,A 0.000,B 0.000,C 90.000,E1 273.037} C_DIS
LIN {X -0.107,Y -491.649,Z 809.514,A 0.000,B 0.000,C 90.000,E1 272.579} C_DIS
LIN {X 0.100,Y -490.591,Z 809.512,A 0.000,B 0.000,C 90.000,E1 272.064} C_DIS
LIN {X -0.170,Y -489.098,Z 809.509,A 0.000,B 0.000,C 90.000,E1 271.604} C_DIS
LIN {X 0.026,Y -487.134,Z 809.506,A 0.000,B 0.000,C 90.000,E1 271.088} C_DIS
LIN {X 0.213,Y -484.713,Z 809.503,A 0.000,B 0.000,C 90.000,E1 270.573} C_DIS
LIN {X -0.099,Y -481.734,Z 809.501,A 0.000,B 0.000,C 90.000,E1 270.115} C_DIS
LIN {X 0.055,Y -478.031,Z 809.498,A 0.000,B 0.000,C 90.000,E1 269.599} C_DIS
LIN {X 0.188,Y -473.504,Z 809.495,A 0.000,B 0.000,C 90.000,E1 269.083} C_DIS
LIN {X -0.175,Y -467.919,Z 809.492,A 0.000,B 0.000,C 90.000,E1 268.625} C_DIS
LIN {X -0.133,Y -464.994,Z 809.491,A 0.000,B 0.000,C 90.000,E1 268.396} C_DIS
LIN {X -0.201,Y -458.537,Z 809.489,A 0.000,B 0.000,C 90.000,E1 267.993} C_DIS
LIN {X 0.132,Y -454.993,Z 809.488,A 0.000,B 0.000,C 90.000,E1 267.764} C_DIS
LIN {X -0.194,Y -451.556,Z 809.487,A 0.000,B 0.000,C 90.000,E1 267.650} C_DIS
LIN {X -0.085,Y -443.766,Z 809.485,A 0.000,B 0.000,C 90.000,E1 267.364} C_DIS
LIN {X 0.104,Y -435.979,Z 809.484,A 0.000,B 0.000,C 90.000,E1 267.135} C_DIS
LIN {X -0.035,Y -428.432,Z 809.483,A 0.000,B 0.000,C 90.000,E1 267.020} C_DIS
LIN {X -0.034,Y -422.626,Z 809.483,A 0.000,B 0.000,C 90.000,E1 266.963} C_DIS
LIN {X -0.103,Y -419.597,Z 809.483,A 0.000,B 0.000,C 90.000,E1 266.963} C_DIS
LIN {X -0.075,Y -180.986,Z 809.483,A 0.000,B 0.000,C 90.000,E1 266.963} C_DIS
LIN {X 0.038,Y -180.838,Z 809.472,A 0.000,B 0.000,C 90.000,E1 264.894} C_DIS
LIN {X -0.059,Y -178.945,Z 809.444,A 0.000,B 0.000,C 90.000,E1 259.859} C_DIS
LIN {X 0.037,Y -176.399,Z 809.420,A 0.000,B 0.000,C 90.000,E1 255.589} C_DIS
LIN {X -0.069,Y -175.503,Z 809.411,A 0.000,B 0.000,C 90.000,E1 253.921} C_DIS
LIN {X -0.007,Y -172.244,Z 809.387,A 0.000,B 0.000,C 90.000,E1 249.625} C_DIS
LIN {X -0.028,Y -171.723,Z 809.382,A 0.000,B 0.000,C 90.000,E1 248.773} C_DIS
LIN {X -0.019,Y -167.318,Z 809.353,A 0.000,B 0.000,C 90.000,E1 243.589} C_DIS
LIN {X -0.086,Y -166.700,Z 809.348,A 0.000,B 0.000,C 90.000,E1 242.743} C_DIS
LIN {X 0.052,Y -162.681,Z 809.324,A 0.000,B 0.000,C 90.000,E1 238.329} C_DIS
LIN {X 0.025,Y -161.371,Z 809.314,A 0.000,B 0.000,C 90.000,E1 236.580} C_DIS
LIN {X -0.066,Y -157.365,Z 809.290,A 0.000,B 0.000,C 90.000,E1 232.190} C_DIS
LIN {X 0.086,Y -155.355,Z 809.275,A 0.000,B 0.000,C 90.000,E1 229.461} C_DIS
LIN {X 0.016,Y -151.699,Z 809.250,A 0.000,B 0.000,C 90.000,E1 225.000} C_DIS
LIN {X -0.046,Y -150.560,Z 809.240,A 0.000,B 0.000,C 90.000,E1 223.218} C_DIS
LIN {X -0.020,Y -147.287,Z 809.215,A 0.000,B 0.000,C 90.000,E1 218.669} C_DIS
LIN {X -0.051,Y -145.316,Z 809.194,A 0.000,B 0.000,C 90.000,E1 215.025} C_DIS
LIN {X -0.011,Y -142.404,Z 809.164,A 0.000,B 0.000,C 90.000,E1 209.489} C_DIS
LIN {X 0.042,Y -141.386,Z 809.148,A 0.000,B 0.000,C 90.000,E1 206.693} C_DIS
LIN {X 0.034,Y -139.350,Z 809.112,A 0.000,B 0.000,C 90.000,E1 200.194} C_DIS
LIN {X 0.024,Y -138.789,Z 809.097,A 0.000,B 0.000,C 90.000,E1 197.402} C_DIS
LIN {X -0.054,Y -138.345,Z 809.055,A 0.000,B 0.000,C 90.000,E1 189.962} C_DIS
LIN {X -0.036,Y -139.384,Z 809.008,A 0.000,B 0.000,C 90.000,E1 181.547} C_DIS
LIN {X 0.017,Y -141.277,Z 808.972,A 0.000,B 0.000,C 90.000,E1 175.008} C_DIS
LIN {X -0.025,Y -142.643,Z 808.957,A 0.000,B 0.000,C 90.000,E1 172.243} C_DIS
LIN {X -0.074,Y -144.975,Z 808.931,A 0.000,B 0.000,C 90.000,E1 167.645} C_DIS
LIN {X 0.058,Y -147.603,Z 808.911,A 0.000,B 0.000,C 90.000,E1 163.921} C_DIS
LIN {X -0.004,Y -150.223,Z 808.891,A 0.000,B 0.000,C 90.000,E1 160.296} C_DIS
LIN {X 0.011,Y -153.612,Z 808.870,A 0.000,B 0.000,C 90.000,E1 156.666} C_DIS
LIN {X 0.000,Y -157.028,Z 808.850,A 0.000,B 0.000,C 90.000,E1 153.076} C_DIS
LIN {X -0.069,Y -161.151,Z 808.831,A 0.000,B 0.000,C 90.000,E1 149.537} C_DIS
LIN {X 0.013,Y -163.249,Z 808.821,A 0.000,B 0.000,C 90.000,E1 147.740} C_DIS
LIN {X -0.023,Y -167.685,Z 808.801,A 0.000,B 0.000,C 90.000,E1 144.242} C_DIS
LIN {X 0.026,Y -171.507,Z 808.787,A 0.000,B 0.000,C 90.000,E1 141.618} C_DIS
LIN {X 0.069,Y -176.442,Z 808.768,A 0.000,B 0.000,C 90.000,E1 138.162} C_DIS
LIN {X -0.059,Y -180.737,Z 808.753,A 0.000,B 0.000,C 90.000,E1 135.648} C_DIS
LIN {X -0.079,Y -186.142,Z 808.735,A 0.000,B 0.000,C 90.000,E1 132.285} C_DIS
LIN {X -0.022,Y -190.781,Z 808.721,A 0.000,B 0.000,C 90.000,E1 129.769} C_DIS
LIN {X -0.029,Y -192.682,Z 808.715,A 0.000,B 0.000,C 90.000,E1 128.624} C_DIS
LIN {X -0.092,Y -293.393,Z 808.714,A 0.000,B 0.000,C 90.000,E1 128.624} C_DIS
LIN {X -0.149,Y -299.327,Z 808.713,A 0.000,B 0.000,C 90.000,E1 128.382} C_DIS
LIN {X 0.078,Y -302.026,Z 808.712,A 0.000,B 0.000,C 90.000,E1 128.096} C_DIS
LIN {X -0.071,Y -305.782,Z 808.709,A 0.000,B 0.000,C 90.000,E1 127.604} C_DIS
LIN {X 0.128,Y -307.438,Z 808.707,A 0.000,B 0.000,C 90.000,E1 127.237} C_DIS
LIN {X -0.104,Y -308.737,Z 808.705,A 0.000,B 0.000,C 90.000,E1 126.950} C_DIS
LIN {X 0.040,Y -320.855,Z 808.684,A 0.000,B 0.000,C 90.000,E1 123.038} C_DIS
LIN {X -0.099,Y -331.330,Z 808.668,A 0.000,B 0.000,C 90.000,E1 120.207} C_DIS
LIN {X 0.008,Y -343.165,Z 808.652,A 0.000,B 0.000,C 90.000,E1 117.385} C_DIS
LIN {X -0.015,Y -356.459,Z 808.637,A 0.000,B 0.000,C 90.000,E1 114.643} C_DIS
LIN {X -0.048,Y -369.600,Z 808.624,A 0.000,B 0.000,C 90.000,E1 112.259} C_DIS
LIN {X -0.175,Y -384.085,Z 808.611,A 0.000,B 0.000,C 90.000,E1 109.939} C_DIS
LIN {X -0.062,Y -400.015,Z 808.598,A 0.000,B 0.000,C 90.000,E1 107.638} C_DIS
LIN {X -0.181,Y -417.508,Z 808.586,A 0.000,B 0.000,C 90.000,E1 105.426} C_DIS
LIN {X -0.064,Y -436.662,Z 808.574,A 0.000,B 0.000,C 90.000,E1 103.244} C_DIS
LIN {X 0.190,Y -456.803,Z 808.562,A 0.000,B 0.000,C 90.000,E1 101.186} C_DIS
LIN {X 0.061,Y -467.080,Z 808.557,A 0.000,B 0.000,C 90.000,E1 100.254} C_DIS
LIN {X 0.090,Y -469.282,Z 808.556,A 0.000,B 0.000,C 90.000,E1 100.018} C_DIS
LIN {X -0.144,Y -471.082,Z 808.554,A 0.000,B 0.000,C 90.000,E1 99.792} C_DIS
LIN {X 0.168,Y -472.432,Z 808.553,A 0.000,B 0.000,C 90.000,E1 99.500} C_DIS
LIN {X -0.118,Y -474.128,Z 808.550,A 0.000,B 0.000,C 90.000,E1 99.029} C_DIS
LIN {X -0.005,Y -474.751,Z 808.547,A 0.000,B 0.000,C 90.000,E1 98.511} C_DIS
LIN {X 0.120,Y -474.411,Z 808.544,A 0.000,B 0.000,C 90.000,E1 97.992} C_DIS
LIN {X -0.219,Y -473.056,Z 808.542,A 0.000,B 0.000,C 90.000,E1 97.530} C_DIS
LIN {X 0.110,Y -471.932,Z 808.540,A 0.000,B 0.000,C 90.000,E1 97.239} C_DIS
LIN {X 0.080,Y -467.110,Z 808.536,A 0.000,B 0.000,C 90.000,E1 96.486} C_DIS
LIN {X 0.061,Y -449.824,Z 808.520,A 0.000,B 0.000,C 90.000,E1 93.669} C_DIS
LIN {X 0.105,Y -439.221,Z 808.510,A 0.000,B 0.000,C 90.000,E1 91.835} C_DIS
LIN {X -0.211,Y -429.892,Z 808.501,A 0.000,B 0.000,C 90.000,E1 90.286} C_DIS
LIN {X 0.156,Y -420.273,Z 808.492,A 0.000,B 0.000,C 90.000,E1 88.625} C_DIS
LIN {X -0.064,Y -410.578,Z 808.483,A 0.000,B 0.000,C 90.000,E1 87.020} C_DIS
LIN {X 0.057,Y -398.980,Z 808.473,A 0.000,B 0.000,C 90.000,E1 85.065} C_DIS
LIN {X -0.014,Y -385.951,Z 808.460,A 0.000,B 0.000,C 90.000,E1 82.818} C_DIS
LIN {X 0.093,Y -371.678,Z 808.446,A 0.000,B 0.000,C 90.000,E1 80.208} C_DIS
LIN {X -0.127,Y -357.939,Z 808.431,A 0.000,B 0.000,C 90.000,E1 77.589} C_DIS
LIN {X -0.066,Y -346.253,Z 808.418,A 0.000,B 0.000,C 90.000,E1 75.172} C_DIS
LIN {X 0.004,Y -336.035,Z 808.406,A 0.000,B 0.000,C 90.000,E1 73.015} C_DIS
LIN {X 0.124,Y -324.581,Z 808.392,A 0.000,B 0.000,C 90.000,E1 70.496} C_DIS
LIN {X -0.020,Y -313.469,Z 808.378,A 0.000,B 0.000,C 90.000,E1 67.975} C_DIS
LIN {X -0.106,Y -298.981,Z 808.358,A 0.000,B 0.000,C 90.000,E1 64.409} C_DIS
LIN {X -0.001,Y -286.749,Z 808.339,A 0.000,B 0.000,C 90.000,E1 61.051} C_DIS
LIN {X -0.105,Y -275.173,Z 808.320,A 0.000,B 0.000,C 90.000,E1 57.661} C_DIS
LIN {X 0.112,Y -265.280,Z 808.303,A 0.000,B 0.000,C 90.000,E1 54.482} C_DIS
LIN {X -0.095,Y -256.711,Z 808.287,A 0.000,B 0.000,C 90.000,E1 51.698} C_DIS
LIN {X 0.123,Y -248.272,Z 808.271,A 0.000,B 0.000,C 90.000,E1 48.771} C_DIS
LIN {X -0.112,Y -238.414,Z 808.251,A 0.000,B 0.000,C 90.000,E1 45.162} C_DIS
LIN {X 0.031,Y -229.338,Z 808.230,A 0.000,B 0.000,C 90.000,E1 41.391} C_DIS
LIN {X -0.090,Y -222.367,Z 808.213,A 0.000,B 0.000,C 90.000,E1 38.382} C_DIS
LIN {X 0.046,Y -213.969,Z 808.192,A 0.000,B 0.000,C 90.000,E1 34.485} C_DIS
LIN {X 0.077,Y -207.872,Z 808.174,A 0.000,B 0.000,C 90.000,E1 31.337} C_DIS
LIN {X -0.006,Y -202.343,Z 808.157,A 0.000,B 0.000,C 90.000,E1 28.180} C_DIS
LIN {X 0.034,Y -197.544,Z 808.139,A 0.000,B 0.000,C 90.000,E1 24.951} C_DIS
LIN {X -0.087,Y -192.676,Z 808.116,A 0.000,B 0.000,C 90.000,E1 20.918} C_DIS
LIN {X -0.074,Y -188.833,Z 808.093,A 0.000,B 0.000,C 90.000,E1 16.804} C_DIS
LIN {X -0.072,Y -185.857,Z 808.066,A 0.000,B 0.000,C 90.000,E1 11.827} C_DIS
LIN {X -0.084,Y -186.376,Z 807.970,A 0.000,B 0.000,C 90.000,E1 354.546} C_DIS
LIN {X 0.075,Y -189.510,Z 807.942,A 0.000,B 0.000,C 90.000,E1 349.511} C_DIS
LIN {X -0.006,Y -193.034,Z 807.919,A 0.000,B 0.000,C 90.000,E1 345.408} C_DIS
LIN {X -0.054,Y -197.469,Z 807.896,A 0.000,B 0.000,C 90.000,E1 341.329} C_DIS
LIN {X 0.116,Y -202.851,Z 807.874,A 0.000,B 0.000,C 90.000,E1 337.230} C_DIS
LIN {X -0.067,Y -207.840,Z 807.856,A 0.000,B 0.000,C 90.000,E1 334.076} C_DIS
LIN {X 0.051,Y -213.518,Z 807.838,A 0.000,B 0.000,C 90.000,E1 330.873} C_DIS
LIN {X 0.068,Y -221.388,Z 807.817,A 0.000,B 0.000,C 90.000,E1 326.962} C_DIS
LIN {X 0.027,Y -230.008,Z 807.795,A 0.000,B 0.000,C 90.000,E1 323.130} C_DIS
LIN {X -0.066,Y -239.391,Z 807.774,A 0.000,B 0.000,C 90.000,E1 319.380} C_DIS
LIN {X 0.097,Y -249.803,Z 807.754,A 0.000,B 0.000,C 90.000,E1 315.648} C_DIS
LIN {X 0.044,Y -259.984,Z 807.736,A 0.000,B 0.000,C 90.000,E1 312.405} C_DIS
LIN {X 0.123,Y -270.866,Z 807.718,A 0.000,B 0.000,C 90.000,E1 309.197} C_DIS
LIN {X 0.158,Y -284.062,Z 807.699,A 0.000,B 0.000,C 90.000,E1 305.724} C_DIS
LIN {X 0.193,Y -298.841,Z 807.680,A 0.000,B 0.000,C 90.000,E1 302.339} C_DIS
LIN {X -0.031,Y -311.925,Z 807.665,A 0.000,B 0.000,C 90.000,E1 299.745} C_DIS
LIN {X -0.145,Y -328.303,Z 807.649,A 0.000,B 0.000,C 90.000,E1 296.873} C_DIS
LIN {X 0.074,Y -347.998,Z 807.632,A 0.000,B 0.000,C 90.000,E1 293.718} C_DIS
LIN {X 0.200,Y -365.518,Z 807.618,A 0.000,B 0.000,C 90.000,E1 291.280} C_DIS
LIN {X -0.062,Y -382.400,Z 807.607,A 0.000,B 0.000,C 90.000,E1 289.268} C_DIS
LIN {X 0.008,Y -402.542,Z 807.594,A 0.000,B 0.000,C 90.000,E1 286.985} C_DIS
LIN {X 0.167,Y -415.065,Z 807.587,A 0.000,B 0.000,C 90.000,E1 285.607} C_DIS
LIN {X 0.165,Y -427.533,Z 807.579,A 0.000,B 0.000,C 90.000,E1 284.245} C_DIS
LIN {X -0.105,Y -439.711,Z 807.572,A 0.000,B 0.000,C 90.000,E1 282.939} C_DIS
LIN {X -0.115,Y -449.043,Z 807.566,A 0.000,B 0.000,C 90.000,E1 281.883} C_DIS
LIN {X -0.102,Y -457.739,Z 807.560,A 0.000,B 0.000,C 90.000,E1 280.838} C_DIS
LIN {X 0.023,Y -465.792,Z 807.554,A 0.000,B 0.000,C 90.000,E1 279.792} C_DIS
LIN {X -0.220,Y -473.190,Z 807.549,A 0.000,B 0.000,C 90.000,E1 278.803} C_DIS
LIN {X 0.221,Y -478.130,Z 807.545,A 0.000,B 0.000,C 90.000,E1 277.992} C_DIS
LIN {X 0.239,Y -482.364,Z 807.540,A 0.000,B 0.000,C 90.000,E1 277.239} C_DIS
LIN {X -0.197,Y -485.991,Z 807.536,A 0.000,B 0.000,C 90.000,E1 276.543} C_DIS
LIN {X -0.058,Y -488.020,Z 807.533,A 0.000,B 0.000,C 90.000,E1 276.030} C_DIS
LIN {X 0.144,Y -489.652,Z 807.531,A 0.000,B 0.000,C 90.000,E1 275.511} C_DIS
LIN {X -0.132,Y -491.011,Z 807.528,A 0.000,B 0.000,C 90.000,E1 275.049} C_DIS
LIN {X 0.088,Y -491.912,Z 807.525,A 0.000,B 0.000,C 90.000,E1 274.531} C_DIS
LIN {X -0.177,Y -492.446,Z 807.523,A 0.000,B 0.000,C 90.000,E1 274.069} C_DIS
LIN {X 0.021,Y -492.575,Z 807.520,A 0.000,B 0.000,C 90.000,E1 273.555} C_DIS
LIN {X 0.251,Y -492.330,Z 807.517,A 0.000,B 0.000,C 90.000,E1 273.037} C_DIS
LIN {X -0.034,Y -491.678,Z 807.514,A 0.000,B 0.000,C 90.000,E1 272.579} C_DIS
LIN {X 0.172,Y -490.630,Z 807.512,A 0.000,B 0.000,C 90.000,E1 272.064} C_DIS
LIN {X -0.099,Y -489.156,Z 807.509,A 0.000,B 0.000,C 90.000,E1 271.604} C_DIS
LIN {X 0.098,Y -487.239,Z 807.506,A 0.000,B 0.000,C 90.000,E1 271.088} C_DIS
LIN {X -0.199,Y -484.836,Z 807.503,A 0.000,B 0.000,C 90.000,E1 270.630} C_DIS
LIN {X -0.027,Y -481.922,Z 807.501,A 0.000,B 0.000,C 90.000,E1 270.115} C_DIS
LIN {X 0.128,Y -478.274,Z 807.498,A 0.000,B 0.000,C 90.000,E1 269.599} C_DIS
LIN {X -0.213,Y -473.811,Z 807.495,A 0.000,B 0.000,C 90.000,E1 269.141} C_DIS
LIN {X -0.101,Y -468.296,Z 807.492,A 0.000,B 0.000,C 90.000,E1 268.625} C_DIS
LIN {X -0.052,Y -462.096,Z 807.490,A 0.000,B 0.000,C 90.000,E1 268.165} C_DIS
LIN {X 0.058,Y -455.261,Z 807.488,A 0.000,B 0.000,C 90.000,E1 267.764} C_DIS
LIN {X 0.171,Y -451.832,Z 807.487,A 0.000,B 0.000,C 90.000,E1 267.593} C_DIS
LIN {X -0.165,Y -447.753,Z 807.486,A 0.000,B 0.000,C 90.000,E1 267.478} C_DIS
LIN {X -0.220,Y -439.850,Z 807.485,A 0.000,B 0.000,C 90.000,E1 267.249} C_DIS
LIN {X 0.173,Y -431.641,Z 807.484,A 0.000,B 0.000,C 90.000,E1 267.020} C_DIS
LIN {X -0.030,Y -424.950,Z 807.483,A 0.000,B 0.000,C 90.000,E1 266.963} C_DIS
LIN {X 0.175,Y -420.334,Z 807.483,A 0.000,B 0.000,C 90.000,E1 266.906} C_DIS
LIN {X 0.045,Y -180.983,Z 807.483,A 0.000,B 0.000,C 90.000,E1 266.906} C_DIS
LIN {X -0.024,Y -180.832,Z 807.472,A 0.000,B 0.000,C 90.000,E1 264.894} C_DIS
LIN {X 0.056,Y -178.939,Z 807.443,A 0.000,B 0.000,C 90.000,E1 259.803} C_DIS
LIN {X -0.077,Y -175.988,Z 807.415,A 0.000,B 0.000,C 90.000,E1 254.755} C_DIS
LIN {X 0.038,Y -175.487,Z 807.410,A 0.000,B 0.000,C 90.000,E1 253.866} C_DIS
LIN {X 0.094,Y -172.231,Z 807.387,A 0.000,B 0.000,C 90.000,E1 249.571} C_DIS
LIN {X 0.072,Y -171.709,Z 807.382,A 0.000,B 0.000,C 90.000,E1 248.720} C_DIS
LIN {X -0.004,Y -167.303,Z 807.353,A 0.000,B 0.000,C 90.000,E1 243.563} C_DIS
LIN {X 0.002,Y -166.683,Z 807.348,A 0.000,B 0.000,C 90.000,E1 242.692} C_DIS
LIN {X -0.007,Y -162.664,Z 807.324,A 0.000,B 0.000,C 90.000,E1 238.329} C_DIS
LIN {X -0.033,Y -161.354,Z 807.314,A 0.000,B 0.000,C 90.000,E1 236.580} C_DIS
LIN {X 0.001,Y -157.348,Z 807.290,A 0.000,B 0.000,C 90.000,E1 232.145} C_DIS
LIN {X 0.030,Y -155.335,Z 807.275,A 0.000,B 0.000,C 90.000,E1 229.461} C_DIS
LIN {X -0.040,Y -151.684,Z 807.250,A 0.000,B 0.000,C 90.000,E1 225.000} C_DIS
LIN {X 0.008,Y -150.548,Z 807.240,A 0.000,B 0.000,C 90.000,E1 223.176} C_DIS
LIN {X 0.040,Y -147.274,Z 807.215,A 0.000,B 0.000,C 90.000,E1 218.624} C_DIS
LIN {X 0.013,Y -145.302,Z 807.194,A 0.000,B 0.000,C 90.000,E1 214.978} C_DIS
LIN {X 0.005,Y -142.395,Z 807.164,A 0.000,B 0.000,C 90.000,E1 209.461} C_DIS
LIN {X -0.012,Y -141.376,Z 807.148,A 0.000,B 0.000,C 90.000,E1 206.693} C_DIS
LIN {X 0.029,Y -139.347,Z 807.112,A 0.000,B 0.000,C 90.000,E1 200.174} C_DIS
LIN {X -0.029,Y -138.784,Z 807.097,A 0.000,B 0.000,C 90.000,E1 197.402} C_DIS
LIN {X 0.030,Y -138.343,Z 807.055,A 0.000,B 0.000,C 90.000,E1 189.905} C_DIS
LIN {X 0.050,Y -139.389,Z 807.008,A 0.000,B 0.000,C 90.000,E1 181.489} C_DIS
LIN {X -0.037,Y -141.287,Z 806.972,A 0.000,B 0.000,C 90.000,E1 175.008} C_DIS
LIN {X 0.063,Y -142.651,Z 806.957,A 0.000,B 0.000,C 90.000,E1 172.186} C_DIS
LIN {X 0.012,Y -144.989,Z 806.931,A 0.000,B 0.000,C 90.000,E1 167.589} C_DIS
LIN {X 0.003,Y -147.616,Z 806.911,A 0.000,B 0.000,C 90.000,E1 163.921} C_DIS
LIN {X 0.081,Y -150.241,Z 806.890,A 0.000,B 0.000,C 90.000,E1 160.242} C_DIS
LIN {X -0.045,Y -153.635,Z 806.870,A 0.000,B 0.000,C 90.000,E1 156.666} C_DIS
LIN {X 0.012,Y -157.050,Z 806.850,A 0.000,B 0.000,C 90.000,E1 153.050} C_DIS
LIN {X 0.011,Y -161.178,Z 806.831,A 0.000,B 0.000,C 90.000,E1 149.488} C_DIS
LIN {X 0.042,Y -163.272,Z 806.821,A 0.000,B 0.000,C 90.000,E1 147.709} C_DIS
LIN {X 0.052,Y -167.714,Z 806.801,A 0.000,B 0.000,C 90.000,E1 144.196} C_DIS
LIN {X -0.035,Y -171.534,Z 806.787,A 0.000,B 0.000,C 90.000,E1 141.618} C_DIS
LIN {X 0.008,Y -176.474,Z 806.768,A 0.000,B 0.000,C 90.000,E1 138.162} C_DIS
LIN {X 0.007,Y -180.771,Z 806.753,A 0.000,B 0.000,C 90.000,E1 135.607} C_DIS
LIN {X -0.006,Y -186.177,Z 806.735,A 0.000,B 0.000,C 90.000,E1 132.243} C_DIS
LIN {X 0.060,Y -190.815,Z 806.721,A 0.000,B 0.000,C 90.000,E1 129.725} C_DIS
LIN {X 0.016,Y -192.660,Z 806.715,A 0.000,B 0.000,C 90.000,E1 128.624} C_DIS
LIN {X -0.011,Y -292.952,Z 806.715,A 0.000,B 0.000,C 90.000,E1 128.624} C_DIS
LIN {X -0.054,Y -295.151,Z 806.714,A 0.000,B 0.000,C 90.000,E1 128.588} C_DIS
LIN {X -0.015,Y -299.674,Z 806.713,A 0.000,B 0.000,C 90.000,E1 128.338} C_DIS
LIN {X -0.024,Y -302.252,Z 806.712,A 0.000,B 0.000,C 90.000,E1 128.096} C_DIS
LIN {X 0.147,Y -306.011,Z 806.709,A 0.000,B 0.000,C 90.000,E1 127.523} C_DIS
LIN {X -0.083,Y -307.605,Z 806.707,A 0.000,B 0.000,C 90.000,E1 127.237} C_DIS
LIN {X 0.117,Y -308.857,Z 806.705,A 0.000,B 0.000,C 90.000,E1 126.870} C_DIS
LIN {X 0.193,Y -319.878,Z 806.685,A 0.000,B 0.000,C 90.000,E1 123.293} C_DIS
LIN {X 0.021,Y -330.227,Z 806.669,A 0.000,B 0.000,C 90.000,E1 120.463} C_DIS
LIN {X 0.102,Y -341.923,Z 806.654,A 0.000,B 0.000,C 90.000,E1 117.641} C_DIS
LIN {X 0.042,Y -355.071,Z 806.638,A 0.000,B 0.000,C 90.000,E1 114.899} C_DIS
LIN {X -0.021,Y -368.071,Z 806.625,A 0.000,B 0.000,C 90.000,E1 112.514} C_DIS
LIN {X -0.049,Y -382.404,Z 806.612,A 0.000,B 0.000,C 90.000,E1 110.174} C_DIS
LIN {X 0.020,Y -398.170,Z 806.599,A 0.000,B 0.000,C 90.000,E1 107.873} C_DIS
LIN {X -0.144,Y -415.486,Z 806.587,A 0.000,B 0.000,C 90.000,E1 105.662} C_DIS
LIN {X 0.001,Y -434.475,Z 806.575,A 0.000,B 0.000,C 90.000,E1 103.467} C_DIS
LIN {X -0.001,Y -454.554,Z 806.563,A 0.000,B 0.000,C 90.000,E1 101.422} C_DIS
LIN {X -0.174,Y -467.363,Z 806.557,A 0.000,B 0.000,C 90.000,E1 100.254} C_DIS
LIN {X -0.144,Y -469.493,Z 806.556,A 0.000,B 0.000,C 90.000,E1 100.018} C_DIS
LIN {X 0.168,Y -471.242,Z 806.554,A 0.000,B 0.000,C 90.000,E1 99.726} C_DIS
LIN {X -0.064,Y -472.556,Z 806.553,A 0.000,B 0.000,C 90.000,E1 99.500} C_DIS
LIN {X 0.117,Y -474.194,Z 806.550,A 0.000,B 0.000,C 90.000,E1 98.973} C_DIS
LIN {X -0.238,Y -474.771,Z 806.547,A 0.000,B 0.000,C 90.000,E1 98.511} C_DIS
LIN {X -0.113,Y -474.384,Z 806.544,A 0.000,B 0.000,C 90.000,E1 97.992} C_DIS
LIN {X 0.080,Y -472.977,Z 806.542,A 0.000,B 0.000,C 90.000,E1 97.466} C_DIS
LIN {X -0.121,Y -471.821,Z 806.540,A 0.000,B 0.000,C 90.000,E1 97.239} C_DIS
LIN {X -0.057,Y -463.680,Z 806.533,A 0.000,B 0.000,C 90.000,E1 95.967} C_DIS
LIN {X 0.021,Y -445.141,Z 806.516,A 0.000,B 0.000,C 90.000,E1 92.865} C_DIS
LIN {X -0.199,Y -436.010,Z 806.507,A 0.000,B 0.000,C 90.000,E1 91.318} C_DIS
LIN {X -0.145,Y -426.549,Z 806.498,A 0.000,B 0.000,C 90.000,E1 89.714} C_DIS
LIN {X -0.145,Y -415.328,Z 806.488,A 0.000,B 0.000,C 90.000,E1 87.822} C_DIS
LIN {X -0.034,Y -405.477,Z 806.479,A 0.000,B 0.000,C 90.000,E1 86.159} C_DIS
LIN {X 0.046,Y -392.304,Z 806.466,A 0.000,B 0.000,C 90.000,E1 83.913} C_DIS
LIN {X -0.131,Y -379.431,Z 806.454,A 0.000,B 0.000,C 90.000,E1 81.659} C_DIS
LIN {X -0.186,Y -366.920,Z 806.441,A 0.000,B 0.000,C 90.000,E1 79.342} C_DIS
LIN {X -0.030,Y -353.454,Z 806.426,A 0.000,B 0.000,C 90.000,E1 76.645} C_DIS
LIN {X 0.005,Y -343.271,Z 806.414,A 0.000,B 0.000,C 90.000,E1 74.519} C_DIS
LIN {X -0.012,Y -331.679,Z 806.400,A 0.000,B 0.000,C 90.000,E1 72.054} C_DIS
LIN {X 0.053,Y -318.981,Z 806.385,A 0.000,B 0.000,C 90.000,E1 69.209} C_DIS
LIN {X -0.003,Y -305.383,Z 806.367,A 0.000,B 0.000,C 90.000,E1 65.997} C_DIS
LIN {X 0.156,Y -294.057,Z 806.350,A 0.000,B 0.000,C 90.000,E1 62.999} C_DIS
LIN {X 0.021,Y -283.302,Z 806.333,A 0.000,B 0.000,C 90.000,E1 59.999} C_DIS
LIN {X 0.012,Y -273.104,Z 806.316,A 0.000,B 0.000,C 90.000,E1 56.914} C_DIS
LIN {X -0.022,Y -265.492,Z 806.303,A 0.000,B 0.000,C 90.000,E1 54.482} C_DIS
LIN {X 0.043,Y -259.091,Z 806.291,A 0.000,B 0.000,C 90.000,E1 52.351} C_DIS
LIN {X -0.035,Y -250.621,Z 806.275,A 0.000,B 0.000,C 90.000,E1 49.504} C_DIS
LIN {X -0.005,Y -240.607,Z 806.255,A 0.000,B 0.000,C 90.000,E1 45.850} C_DIS
LIN {X 0.023,Y -231.410,Z 806.234,A 0.000,B 0.000,C 90.000,E1 42.123} C_DIS
LIN {X -0.053,Y -224.379,Z 806.217,A 0.000,B 0.000,C 90.000,E1 39.116} C_DIS
LIN {X 0.097,Y -215.908,Z 806.196,A 0.000,B 0.000,C 90.000,E1 35.231} C_DIS
LIN {X -0.007,Y -209.608,Z 806.179,A 0.000,B 0.000,C 90.000,E1 32.133} C_DIS
LIN {X 0.040,Y -202.619,Z 806.156,A 0.000,B 0.000,C 90.000,E1 28.153} C_DIS
LIN {X -0.007,Y -197.825,Z 806.139,A 0.000,B 0.000,C 90.000,E1 24.951} C_DIS
LIN {X 0.062,Y -192.961,Z 806.116,A 0.000,B 0.000,C 90.000,E1 20.865} C_DIS
LIN {X -0.097,Y -189.123,Z 806.093,A 0.000,B 0.000,C 90.000,E1 16.804} C_DIS
LIN {X -0.084,Y -186.119,Z 806.066,A 0.000,B 0.000,C 90.000,E1 11.827} C_DIS
LIN {X 0.004,Y -186.184,Z 805.974,A 0.000,B 0.000,C 90.000,E1 355.355} C_DIS
LIN {X -0.068,Y -189.088,Z 805.946,A 0.000,B 0.000,C 90.000,E1 350.387} C_DIS
LIN {X 0.026,Y -192.414,Z 805.924,A 0.000,B 0.000,C 90.000,E1 346.228} C_DIS
LIN {X 0.036,Y -196.673,Z 805.901,A 0.000,B 0.000,C 90.000,E1 342.127} C_DIS
LIN {X -0.086,Y -201.851,Z 805.878,A 0.000,B 0.000,C 90.000,E1 338.103} C_DIS
LIN {X -0.029,Y -208.011,Z 805.856,A 0.000,B 0.000,C 90.000,E1 334.076} C_DIS
LIN {X -0.091,Y -213.702,Z 805.838,A 0.000,B 0.000,C 90.000,E1 330.923} C_DIS
LIN {X -0.002,Y -221.565,Z 805.817,A 0.000,B 0.000,C 90.000,E1 326.993} C_DIS
LIN {X 0.085,Y -230.172,Z 805.795,A 0.000,B 0.000,C 90.000,E1 323.130} C_DIS
LIN {X -0.002,Y -239.528,Z 805.774,A 0.000,B 0.000,C 90.000,E1 319.380} C_DIS
LIN {X -0.001,Y -248.852,Z 805.756,A 0.000,B 0.000,C 90.000,E1 316.053} C_DIS
LIN {X 0.086,Y -258.910,Z 805.738,A 0.000,B 0.000,C 90.000,E1 312.771} C_DIS
LIN {X 0.135,Y -269.645,Z 805.720,A 0.000,B 0.000,C 90.000,E1 309.564} C_DIS
LIN {X 0.016,Y -281.324,Z 805.703,A 0.000,B 0.000,C 90.000,E1 306.457} C_DIS
LIN {X -0.121,Y -295.725,Z 805.684,A 0.000,B 0.000,C 90.000,E1 303.086} C_DIS
LIN {X 0.025,Y -310.132,Z 805.667,A 0.000,B 0.000,C 90.000,E1 300.079} C_DIS
LIN {X 0.009,Y -326.305,Z 805.651,A 0.000,B 0.000,C 90.000,E1 297.180} C_DIS
LIN {X -0.150,Y -343.751,Z 805.635,A 0.000,B 0.000,C 90.000,E1 294.387} C_DIS
LIN {X 0.128,Y -358.575,Z 805.623,A 0.000,B 0.000,C 90.000,E1 292.206} C_DIS
LIN {X 0.055,Y -372.364,Z 805.614,A 0.000,B 0.000,C 90.000,E1 290.429} C_DIS
LIN {X -0.107,Y -389.691,Z 805.602,A 0.000,B 0.000,C 90.000,E1 288.417} C_DIS
LIN {X -0.032,Y -409.593,Z 805.590,A 0.000,B 0.000,C 90.000,E1 286.205} C_DIS
LIN {X 0.063,Y -422.127,Z 805.582,A 0.000,B 0.000,C 90.000,E1 284.828} C_DIS
LIN {X -0.107,Y -436.737,Z 805.573,A 0.000,B 0.000,C 90.000,E1 283.244} C_DIS
LIN {X -0.051,Y -446.213,Z 805.568,A 0.000,B 0.000,C 90.000,E1 282.175} C_DIS
LIN {X -0.072,Y -455.105,Z 805.562,A 0.000,B 0.000,C 90.000,E1 281.130} C_DIS
LIN {X 0.103,Y -463.317,Z 805.556,A 0.000,B 0.000,C 90.000,E1 280.074} C_DIS
LIN {X -0.172,Y -470.904,Z 805.550,A 0.000,B 0.000,C 90.000,E1 279.086} C_DIS
LIN {X 0.247,Y -476.139,Z 805.546,A 0.000,B 0.000,C 90.000,E1 278.276} C_DIS
LIN {X 0.177,Y -480.663,Z 805.542,A 0.000,B 0.000,C 90.000,E1 277.530} C_DIS
LIN {X 0.216,Y -484.532,Z 805.538,A 0.000,B 0.000,C 90.000,E1 276.777} C_DIS
LIN {X -0.257,Y -487.770,Z 805.534,A 0.000,B 0.000,C 90.000,E1 276.087} C_DIS
LIN {X -0.051,Y -489.482,Z 805.531,A 0.000,B 0.000,C 90.000,E1 275.568} C_DIS
LIN {X 0.159,Y -490.859,Z 805.528,A 0.000,B 0.000,C 90.000,E1 275.049} C_DIS
LIN {X -0.112,Y -491.804,Z 805.525,A 0.000,B 0.000,C 90.000,E1 274.588} C_DIS
LIN {X 0.079,Y -492.365,Z 805.523,A 0.000,B 0.000,C 90.000,E1 274.073} C_DIS
LIN {X -0.182,Y -492.552,Z 805.520,A 0.000,B 0.000,C 90.000,E1 273.612} C_DIS
LIN {X 0.049,Y -492.330,Z 805.517,A 0.000,B 0.000,C 90.000,E1 273.094} C_DIS
LIN {X -0.237,Y -491.741,Z 805.514,A 0.000,B 0.000,C 90.000,E1 272.636} C_DIS
LIN {X -0.030,Y -490.718,Z 805.512,A 0.000,B 0.000,C 90.000,E1 272.121} C_DIS
LIN {X 0.189,Y -489.314,Z 805.509,A 0.000,B 0.000,C 90.000,E1 271.604} C_DIS
LIN {X -0.103,Y -487.447,Z 805.506,A 0.000,B 0.000,C 90.000,E1 271.146} C_DIS
LIN {X 0.087,Y -485.117,Z 805.504,A 0.000,B 0.000,C 90.000,E1 270.630} C_DIS
LIN {X -0.224,Y -482.253,Z 805.501,A 0.000,B 0.000,C 90.000,E1 270.172} C_DIS
LIN {X -0.066,Y -478.709,Z 805.498,A 0.000,B 0.000,C 90.000,E1 269.656} C_DIS
LIN {X 0.072,Y -474.317,Z 805.495,A 0.000,B 0.000,C 90.000,E1 269.141} C_DIS
LIN {X -0.107,Y -471.803,Z 805.494,A 0.000,B 0.000,C 90.000,E1 268.912} C_DIS
LIN {X 0.183,Y -468.976,Z 805.492,A 0.000,B 0.000,C 90.000,E1 268.625} C_DIS
LIN {X 0.174,Y -462.865,Z 805.490,A 0.000,B 0.000,C 90.000,E1 268.167} C_DIS
LIN {X -0.031,Y -459.694,Z 805.489,A 0.000,B 0.000,C 90.000,E1 267.993} C_DIS
LIN {X 0.209,Y -456.063,Z 805.488,A 0.000,B 0.000,C 90.000,E1 267.764} C_DIS
LIN {X -0.158,Y -452.667,Z 805.487,A 0.000,B 0.000,C 90.000,E1 267.650} C_DIS
LIN {X -0.070,Y -448.671,Z 805.486,A 0.000,B 0.000,C 90.000,E1 267.478} C_DIS
LIN {X -0.194,Y -440.825,Z 805.485,A 0.000,B 0.000,C 90.000,E1 267.249} C_DIS
LIN {X 0.158,Y -432.692,Z 805.484,A 0.000,B 0.000,C 90.000,E1 267.020} C_DIS
LIN {X -0.139,Y -425.576,Z 805.483,A 0.000,B 0.000,C 90.000,E1 266.963} C_DIS
LIN {X -0.011,Y -418.370,Z 805.483,A 0.000,B 0.000,C 90.000,E1 266.906} C_DIS
LIN {X -0.030,Y -180.981,Z 805.483,A 0.000,B 0.000,C 90.000,E1 266.906} C_DIS
LIN {X -0.049,Y -180.891,Z 805.473,A 0.000,B 0.000,C 90.000,E1 265.179} C_DIS
LIN {X 0.013,Y -179.016,Z 805.445,A 0.000,B 0.000,C 90.000,E1 260.095} C_DIS
LIN {X -0.068,Y -178.643,Z 805.440,A 0.000,B 0.000,C 90.000,E1 259.275} C_DIS
LIN {X 0.005,Y -175.695,Z 805.412,A 0.000,B 0.000,C 90.000,E1 254.157} C_DIS
LIN {X 0.017,Y -172.411,Z 805.388,A 0.000,B 0.000,C 90.000,E1 249.880} C_DIS
LIN {X 0.033,Y -171.227,Z 805.379,A 0.000,B 0.000,C 90.000,E1 248.156} C_DIS
LIN {X 0.009,Y -167.507,Z 805.355,A 0.000,B 0.000,C 90.000,E1 243.845} C_DIS
LIN {X -0.058,Y -166.903,Z 805.350,A 0.000,B 0.000,C 90.000,E1 242.999} C_DIS
LIN {X -0.006,Y -162.211,Z 805.321,A 0.000,B 0.000,C 90.000,E1 237.740} C_DIS
LIN {X 0.047,Y -160.787,Z 805.311,A 0.000,B 0.000,C 90.000,E1 235.960} C_DIS
LIN {X 0.018,Y -157.578,Z 805.291,A 0.000,B 0.000,C 90.000,E1 232.431} C_DIS
LIN {X 0.052,Y -155.611,Z 805.276,A 0.000,B 0.000,C 90.000,E1 229.747} C_DIS
LIN {X -0.005,Y -151.889,Z 805.252,A 0.000,B 0.000,C 90.000,E1 225.283} C_DIS
LIN {X -0.096,Y -150.117,Z 805.237,A 0.000,B 0.000,C 90.000,E1 222.609} C_DIS
LIN {X 0.032,Y -146.909,Z 805.211,A 0.000,B 0.000,C 90.000,E1 218.016} C_DIS
LIN {X -0.067,Y -145.497,Z 805.196,A 0.000,B 0.000,C 90.000,E1 215.311} C_DIS
LIN {X 0.052,Y -142.903,Z 805.170,A 0.000,B 0.000,C 90.000,E1 210.669} C_DIS
LIN {X -0.019,Y -141.523,Z 805.150,A 0.000,B 0.000,C 90.000,E1 207.001} C_DIS
LIN {X 0.025,Y -139.396,Z 805.114,A 0.000,B 0.000,C 90.000,E1 200.482} C_DIS
LIN {X 0.076,Y -139.108,Z 805.104,A 0.000,B 0.000,C 90.000,E1 198.598} C_DIS
LIN {X -0.069,Y -138.353,Z 805.057,A 0.000,B 0.000,C 90.000,E1 190.254} C_DIS
LIN {X 0.061,Y -139.510,Z 805.005,A 0.000,B 0.000,C 90.000,E1 180.859} C_DIS
LIN {X 0.001,Y -141.153,Z 804.974,A 0.000,B 0.000,C 90.000,E1 175.298} C_DIS
LIN {X -0.028,Y -142.532,Z 804.958,A 0.000,B 0.000,C 90.000,E1 172.527} C_DIS
LIN {X 0.041,Y -144.800,Z 804.933,A 0.000,B 0.000,C 90.000,E1 167.881} C_DIS
LIN {X 0.029,Y -147.420,Z 804.912,A 0.000,B 0.000,C 90.000,E1 164.212} C_DIS
LIN {X 0.058,Y -149.996,Z 804.892,A 0.000,B 0.000,C 90.000,E1 160.550} C_DIS
LIN {X 0.066,Y -153.325,Z 804.872,A 0.000,B 0.000,C 90.000,E1 156.922} C_DIS
LIN {X -0.023,Y -155.025,Z 804.862,A 0.000,B 0.000,C 90.000,E1 155.153} C_DIS
LIN {X -0.002,Y -158.672,Z 804.842,A 0.000,B 0.000,C 90.000,E1 151.563} C_DIS
LIN {X 0.081,Y -161.951,Z 804.827,A 0.000,B 0.000,C 90.000,E1 148.869} C_DIS
LIN {X -0.035,Y -166.141,Z 804.808,A 0.000,B 0.000,C 90.000,E1 145.388} C_DIS
LIN {X -0.038,Y -171.154,Z 804.788,A 0.000,B 0.000,C 90.000,E1 141.904} C_DIS
LIN {X -0.003,Y -176.032,Z 804.769,A 0.000,B 0.000,C 90.000,E1 138.447} C_DIS
LIN {X -0.008,Y -180.287,Z 804.755,A 0.000,B 0.000,C 90.000,E1 135.891} C_DIS
LIN {X -0.036,Y -185.699,Z 804.736,A 0.000,B 0.000,C 90.000,E1 132.528} C_DIS
LIN {X 0.016,Y -190.303,Z 804.722,A 0.000,B 0.000,C 90.000,E1 130.011} C_DIS
LIN {X 0.054,Y -192.640,Z 804.715,A 0.000,B 0.000,C 90.000,E1 128.624} C_DIS
LIN {X 0.037,Y -292.784,Z 804.715,A 0.000,B 0.000,C 90.000,E1 128.624} C_DIS
LIN {X -0.101,Y -294.449,Z 804.714,A 0.000,B 0.000,C 90.000,E1 128.624} C_DIS
LIN {X -0.104,Y -299.378,Z 804.713,A 0.000,B 0.000,C 90.000,E1 128.382} C_DIS
LIN {X 0.041,Y -302.572,Z 804.711,A 0.000,B 0.000,C 90.000,E1 128.051} C_DIS
LIN {X -0.050,Y -306.211,Z 804.708,A 0.000,B 0.000,C 90.000,E1 127.523} C_DIS
LIN {X 0.151,Y -307.752,Z 804.707,A 0.000,B 0.000,C 90.000,E1 127.156} C_DIS
LIN {X -0.080,Y -308.961,Z 804.705,A 0.000,B 0.000,C 90.000,E1 126.870} C_DIS
LIN {X -0.007,Y -319.977,Z 804.685,A 0.000,B 0.000,C 90.000,E1 123.293} C_DIS
LIN {X -0.181,Y -330.344,Z 804.669,A 0.000,B 0.000,C 90.000,E1 120.463} C_DIS
LIN {X -0.106,Y -342.056,Z 804.653,A 0.000,B 0.000,C 90.000,E1 117.641} C_DIS
LIN {X -0.170,Y -355.223,Z 804.638,A 0.000,B 0.000,C 90.000,E1 114.899} C_DIS
LIN {X 0.104,Y -368.241,Z 804.625,A 0.000,B 0.000,C 90.000,E1 112.461} C_DIS
LIN {X 0.092,Y -382.592,Z 804.612,A 0.000,B 0.000,C 90.000,E1 110.120} C_DIS
LIN {X 0.176,Y -398.380,Z 804.599,A 0.000,B 0.000,C 90.000,E1 107.819} C_DIS
LIN {X 0.028,Y -415.717,Z 804.587,A 0.000,B 0.000,C 90.000,E1 105.607} C_DIS
LIN {X 0.191,Y -434.732,Z 804.575,A 0.000,B 0.000,C 90.000,E1 103.411} C_DIS
LIN {X -0.225,Y -454.818,Z 804.563,A 0.000,B 0.000,C 90.000,E1 101.422} C_DIS
LIN {X 0.068,Y -467.617,Z 804.557,A 0.000,B 0.000,C 90.000,E1 100.197} C_DIS
LIN {X 0.101,Y -469.687,Z 804.555,A 0.000,B 0.000,C 90.000,E1 99.962} C_DIS
LIN {X -0.050,Y -471.394,Z 804.554,A 0.000,B 0.000,C 90.000,E1 99.726} C_DIS
LIN {X 0.185,Y -472.675,Z 804.553,A 0.000,B 0.000,C 90.000,E1 99.443} C_DIS
LIN {X -0.101,Y -474.264,Z 804.550,A 0.000,B 0.000,C 90.000,E1 98.973} C_DIS
LIN {X 0.014,Y -474.800,Z 804.547,A 0.000,B 0.000,C 90.000,E1 98.454} C_DIS
LIN {X 0.141,Y -474.373,Z 804.544,A 0.000,B 0.000,C 90.000,E1 97.936} C_DIS
LIN {X -0.135,Y -472.920,Z 804.541,A 0.000,B 0.000,C 90.000,E1 97.466} C_DIS
LIN {X 0.132,Y -471.735,Z 804.540,A 0.000,B 0.000,C 90.000,E1 97.182} C_DIS
LIN {X 0.069,Y -452.553,Z 804.523,A 0.000,B 0.000,C 90.000,E1 94.131} C_DIS
LIN {X -0.068,Y -440.486,Z 804.511,A 0.000,B 0.000,C 90.000,E1 92.064} C_DIS
LIN {X 0.071,Y -431.177,Z 804.503,A 0.000,B 0.000,C 90.000,E1 90.458} C_DIS
LIN {X 0.154,Y -420.016,Z 804.492,A 0.000,B 0.000,C 90.000,E1 88.568} C_DIS
LIN {X -0.070,Y -410.316,Z 804.483,A 0.000,B 0.000,C 90.000,E1 86.963} C_DIS
LIN {X 0.044,Y -398.761,Z 804.472,A 0.000,B 0.000,C 90.000,E1 85.008} C_DIS
LIN {X 0.011,Y -384.111,Z 804.458,A 0.000,B 0.000,C 90.000,E1 82.470} C_DIS
LIN {X 0.067,Y -371.517,Z 804.445,A 0.000,B 0.000,C 90.000,E1 80.151} C_DIS
LIN {X -0.083,Y -357.798,Z 804.431,A 0.000,B 0.000,C 90.000,E1 77.521} C_DIS
LIN {X -0.016,Y -346.106,Z 804.417,A 0.000,B 0.000,C 90.000,E1 75.102} C_DIS
LIN {X -0.040,Y -335.957,Z 804.405,A 0.000,B 0.000,C 90.000,E1 72.960} C_DIS
LIN {X 0.185,Y -324.537,Z 804.391,A 0.000,B 0.000,C 90.000,E1 70.423} C_DIS
LIN {X -0.072,Y -313.435,Z 804.377,A 0.000,B 0.000,C 90.000,E1 67.922} C_DIS
LIN {X -0.035,Y -299.076,Z 804.357,A 0.000,B 0.000,C 90.000,E1 64.332} C_DIS
LIN {X -0.060,Y -286.949,Z 804.339,A 0.000,B 0.000,C 90.000,E1 61.001} C_DIS
LIN {X -0.015,Y -275.523,Z 804.320,A 0.000,B 0.000,C 90.000,E1 57.582} C_DIS
LIN {X -0.150,Y -265.719,Z 804.302,A 0.000,B 0.000,C 90.000,E1 54.482} C_DIS
LIN {X -0.079,Y -259.339,Z 804.291,A 0.000,B 0.000,C 90.000,E1 52.351} C_DIS
LIN {X 0.045,Y -250.899,Z 804.275,A 0.000,B 0.000,C 90.000,E1 49.461} C_DIS
LIN {X 0.065,Y -240.907,Z 804.255,A 0.000,B 0.000,C 90.000,E1 45.810} C_DIS
LIN {X -0.063,Y -231.720,Z 804.234,A 0.000,B 0.000,C 90.000,E1 42.123} C_DIS
LIN {X 0.046,Y -224.676,Z 804.217,A 0.000,B 0.000,C 90.000,E1 39.072} C_DIS
LIN {X 0.033,Y -216.194,Z 804.196,A 0.000,B 0.000,C 90.000,E1 35.231} C_DIS
LIN {X -0.062,Y -209.885,Z 804.178,A 0.000,B 0.000,C 90.000,E1 32.133} C_DIS
LIN {X -0.003,Y -202.907,Z 804.156,A 0.000,B 0.000,C 90.000,E1 28.153} C_DIS
LIN {X -0.044,Y -198.112,Z 804.139,A 0.000,B 0.000,C 90.000,E1 24.951} C_DIS
LIN {X -0.084,Y -194.117,Z 804.120,A 0.000,B 0.000,C 90.000,E1 21.716} C_DIS
LIN {X 0.033,Y -190.083,Z 804.098,A 0.000,B 0.000,C 90.000,E1 17.583} C_DIS
LIN {X -0.057,Y -186.777,Z 804.070,A 0.000,B 0.000,C 90.000,E1 12.647} C_DIS
LIN {X 0.069,Y -184.581,Z 804.029,A 0.000,B 0.000,C 90.000,E1 5.106} C_DIS
LIN {X 0.010,Y -186.389,Z 803.974,A 0.000,B 0.000,C 90.000,E1 355.355} C_DIS
LIN {X -0.053,Y -189.258,Z 803.947,A 0.000,B 0.000,C 90.000,E1 350.387} C_DIS
LIN {X 0.046,Y -192.586,Z 803.924,A 0.000,B 0.000,C 90.000,E1 346.228} C_DIS
LIN {X 0.061,Y -196.832,Z 803.901,A 0.000,B 0.000,C 90.000,E1 342.127} C_DIS
LIN {X -0.054,Y -202.018,Z 803.878,A 0.000,B 0.000,C 90.000,E1 338.103} C_DIS
LIN {X 0.113,Y -206.862,Z 803.860,A 0.000,B 0.000,C 90.000,E1 334.845} C_DIS
LIN {X 0.026,Y -212.402,Z 803.843,A 0.000,B 0.000,C 90.000,E1 331.691} C_DIS
LIN {X -0.027,Y -220.116,Z 803.821,A 0.000,B 0.000,C 90.000,E1 327.788} C_DIS
LIN {X 0.019,Y -226.795,Z 803.804,A 0.000,B 0.000,C 90.000,E1 324.689} C_DIS
LIN {X 0.046,Y -235.827,Z 803.783,A 0.000,B 0.000,C 90.000,E1 320.884} C_DIS
LIN {X -0.056,Y -244.774,Z 803.764,A 0.000,B 0.000,C 90.000,E1 317.553} C_DIS
LIN {X -0.096,Y -254.453,Z 803.746,A 0.000,B 0.000,C 90.000,E1 314.271} C_DIS
LIN {X -0.152,Y -266.018,Z 803.726,A 0.000,B 0.000,C 90.000,E1 310.701} C_DIS
LIN {X -0.041,Y -277.382,Z 803.708,A 0.000,B 0.000,C 90.000,E1 307.523} C_DIS
LIN {X -0.012,Y -288.309,Z 803.693,A 0.000,B 0.000,C 90.000,E1 304.771} C_DIS
LIN {X 0.001,Y -303.470,Z 803.675,A 0.000,B 0.000,C 90.000,E1 301.416} C_DIS
LIN {X -0.015,Y -315.255,Z 803.662,A 0.000,B 0.000,C 90.000,E1 299.127} C_DIS
LIN {X 0.061,Y -333.805,Z 803.644,A 0.000,B 0.000,C 90.000,E1 295.924} C_DIS
LIN {X -0.035,Y -349.775,Z 803.630,A 0.000,B 0.000,C 90.000,E1 293.462} C_DIS
LIN {X -0.006,Y -367.399,Z 803.617,A 0.000,B 0.000,C 90.000,E1 291.046} C_DIS
LIN {X -0.008,Y -389.417,Z 803.602,A 0.000,B 0.000,C 90.000,E1 288.417} C_DIS
LIN {X -0.055,Y -407.227,Z 803.591,A 0.000,B 0.000,C 90.000,E1 286.441} C_DIS
LIN {X -0.024,Y -419.834,Z 803.584,A 0.000,B 0.000,C 90.000,E1 285.064} C_DIS
LIN {X 0.011,Y -432.177,Z 803.576,A 0.000,B 0.000,C 90.000,E1 283.703} C_DIS
LIN {X 0.129,Y -444.161,Z 803.569,A 0.000,B 0.000,C 90.000,E1 282.355} C_DIS
LIN {X 0.178,Y -453.199,Z 803.563,A 0.000,B 0.000,C 90.000,E1 281.299} C_DIS
LIN {X -0.206,Y -461.539,Z 803.557,A 0.000,B 0.000,C 90.000,E1 280.310} C_DIS
LIN {X -0.039,Y -469.263,Z 803.551,A 0.000,B 0.000,C 90.000,E1 279.265} C_DIS
LIN {X -0.107,Y -474.622,Z 803.547,A 0.000,B 0.000,C 90.000,E1 278.511} C_DIS
LIN {X -0.123,Y -479.371,Z 803.543,A 0.000,B 0.000,C 90.000,E1 277.757} C_DIS
LIN {X -0.104,Y -483.436,Z 803.539,A 0.000,B 0.000,C 90.000,E1 277.004} C_DIS
LIN {X -0.103,Y -486.856,Z 803.535,A 0.000,B 0.000,C 90.000,E1 276.258} C_DIS
LIN {X 0.260,Y -487.862,Z 803.533,A 0.000,B 0.000,C 90.000,E1 275.967} C_DIS
LIN {X -0.070,Y -489.555,Z 803.531,A 0.000,B 0.000,C 90.000,E1 275.511} C_DIS
LIN {X 0.141,Y -490.900,Z 803.528,A 0.000,B 0.000,C 90.000,E1 274.992} C_DIS
LIN {X -0.128,Y -491.825,Z 803.525,A 0.000,B 0.000,C 90.000,E1 274.531} C_DIS
LIN {X 0.097,Y -492.396,Z 803.522,A 0.000,B 0.000,C 90.000,E1 274.012} C_DIS
LIN {X -0.198,Y -492.513,Z 803.520,A 0.000,B 0.000,C 90.000,E1 273.555} C_DIS
LIN {X 0.034,Y -492.260,Z 803.517,A 0.000,B 0.000,C 90.000,E1 273.037} C_DIS
LIN {X 0.238,Y -491.647,Z 803.514,A 0.000,B 0.000,C 90.000,E1 272.522} C_DIS
LIN {X -0.046,Y -490.612,Z 803.511,A 0.000,B 0.000,C 90.000,E1 272.064} C_DIS
LIN {X 0.172,Y -489.171,Z 803.509,A 0.000,B 0.000,C 90.000,E1 271.547} C_DIS
LIN {X -0.119,Y -487.246,Z 803.506,A 0.000,B 0.000,C 90.000,E1 271.088} C_DIS
LIN {X 0.069,Y -484.875,Z 803.503,A 0.000,B 0.000,C 90.000,E1 270.573} C_DIS
LIN {X 0.240,Y -481.940,Z 803.500,A 0.000,B 0.000,C 90.000,E1 270.057} C_DIS
LIN {X -0.084,Y -478.389,Z 803.498,A 0.000,B 0.000,C 90.000,E1 269.599} C_DIS
LIN {X 0.221,Y -476.305,Z 803.496,A 0.000,B 0.000,C 90.000,E1 269.312} C_DIS
LIN {X -0.130,Y -471.370,Z 803.494,A 0.000,B 0.000,C 90.000,E1 268.854} C_DIS
LIN {X 0.175,Y -465.612,Z 803.491,A 0.000,B 0.000,C 90.000,E1 268.339} C_DIS
LIN {X 0.031,Y -459.228,Z 803.489,A 0.000,B 0.000,C 90.000,E1 267.936} C_DIS
LIN {X -0.021,Y -452.215,Z 803.487,A 0.000,B 0.000,C 90.000,E1 267.593} C_DIS
LIN {X 0.041,Y -444.625,Z 803.485,A 0.000,B 0.000,C 90.000,E1 267.306} C_DIS
LIN {X 0.164,Y -436.740,Z 803.484,A 0.000,B 0.000,C 90.000,E1 267.078} C_DIS
LIN {X -0.002,Y -429.192,Z 803.483,A 0.000,B 0.000,C 90.000,E1 266.963} C_DIS
LIN {X -0.109,Y -420.156,Z 803.483,A 0.000,B 0.000,C 90.000,E1 266.906} C_DIS
LIN {X -0.080,Y -180.980,Z 803.483,A 0.000,B 0.000,C 90.000,E1 266.906} C_DIS
LIN {X 0.031,Y -180.820,Z 803.471,A 0.000,B 0.000,C 90.000,E1 264.837} C_DIS
LIN {X -0.069,Y -178.923,Z 803.443,A 0.000,B 0.000,C 90.000,E1 259.803} C_DIS
LIN {X -0.030,Y -175.970,Z 803.415,A 0.000,B 0.000,C 90.000,E1 254.700} C_DIS
LIN {X -0.036,Y -175.453,Z 803.410,A 0.000,B 0.000,C 90.000,E1 253.850} C_DIS
LIN {X -0.028,Y -172.206,Z 803.386,A 0.000,B 0.000,C 90.000,E1 249.571} C_DIS
LIN {X -0.050,Y -171.681,Z 803.382,A 0.000,B 0.000,C 90.000,E1 248.720} C_DIS
LIN {X -0.059,Y -167.908,Z 803.358,A 0.000,B 0.000,C 90.000,E1 244.409} C_DIS
LIN {X -0.041,Y -166.648,Z 803.348,A 0.000,B 0.000,C 90.000,E1 242.666} C_DIS
LIN {X 0.014,Y -162.632,Z 803.324,A 0.000,B 0.000,C 90.000,E1 238.280} C_DIS
LIN {X 0.073,Y -161.320,Z 803.314,A 0.000,B 0.000,C 90.000,E1 236.501} C_DIS
LIN {X -0.018,Y -157.315,Z 803.289,A 0.000,B 0.000,C 90.000,E1 232.110} C_DIS
LIN {X -0.085,Y -155.295,Z 803.275,A 0.000,B 0.000,C 90.000,E1 229.461} C_DIS
LIN {X 0.062,Y -151.655,Z 803.250,A 0.000,B 0.000,C 90.000,E1 224.919} C_DIS
LIN {X -0.001,Y -150.523,Z 803.240,A 0.000,B 0.000,C 90.000,E1 223.137} C_DIS
LIN {X 0.023,Y -147.248,Z 803.214,A 0.000,B 0.000,C 90.000,E1 218.588} C_DIS
LIN {X -0.013,Y -145.273,Z 803.194,A 0.000,B 0.000,C 90.000,E1 214.945} C_DIS
LIN {X 0.021,Y -142.379,Z 803.163,A 0.000,B 0.000,C 90.000,E1 209.411} C_DIS
LIN {X 0.070,Y -141.355,Z 803.148,A 0.000,B 0.000,C 90.000,E1 206.616} C_DIS
LIN {X 0.053,Y -139.341,Z 803.112,A 0.000,B 0.000,C 90.000,E1 200.120} C_DIS
LIN {X -0.028,Y -139.009,Z 803.102,A 0.000,B 0.000,C 90.000,E1 198.290} C_DIS
LIN {X 0.059,Y -138.340,Z 803.055,A 0.000,B 0.000,C 90.000,E1 189.849} C_DIS
LIN {X -0.057,Y -139.402,Z 803.008,A 0.000,B 0.000,C 90.000,E1 181.489} C_DIS
LIN {X -0.004,Y -141.308,Z 802.972,A 0.000,B 0.000,C 90.000,E1 174.951} C_DIS
LIN {X -0.046,Y -142.668,Z 802.956,A 0.000,B 0.000,C 90.000,E1 172.186} C_DIS
LIN {X 0.075,Y -145.017,Z 802.931,A 0.000,B 0.000,C 90.000,E1 167.521} C_DIS
LIN {X 0.033,Y -147.643,Z 802.910,A 0.000,B 0.000,C 90.000,E1 163.866} C_DIS
LIN {X -0.031,Y -150.276,Z 802.890,A 0.000,B 0.000,C 90.000,E1 160.242} C_DIS
LIN {X -0.018,Y -153.679,Z 802.870,A 0.000,B 0.000,C 90.000,E1 156.613} C_DIS
LIN {X 0.037,Y -157.094,Z 802.850,A 0.000,B 0.000,C 90.000,E1 152.999} C_DIS
END
